LIN {X 0,Y 282.677,Z 621.959,A -85,B 0,C 180,E1 -17002.141,E2 -17002.141} C_VEL
LIN {X 0,Y 282.367,Z 625.254,A -85,B 0,C 180,E1 -17004.621,E2 -17004.621} C_VEL
LIN {X 0,Y 282.315,Z 626.398,A -85,B 0,C 180,E1 -17005.718,E2 -17005.718} C_VEL
LIN {X 0,Y 282.332,Z 627.925,A -85,B 0,C 180,E1 -17008.574,E2 -17008.574} C_VEL
LIN {X 0,Y 282.345,Z 628.204,A -85,B 0,C 180,E1 -17010,E2 -17010} C_VEL
LIN {X 0,Y 282.337,Z 627.328,A -85,B 0,C 180,E1 -17012.854,E2 -17012.854} C_VEL
LIN {X 0,Y 282.306,Z 626.397,A -85,B 0,C 180,E1 -17014.283,E2 -17014.283} C_VEL
LIN {X 0,Y 282.519,Z 623.046,A -85,B 0,C 180,E1 -17017.145,E2 -17017.145} C_VEL
LIN {X 0,Y 282.977,Z 619.419,A -85,B 0,C 180,E1 -17019.29,E2 -17019.29} C_VEL
LIN {X 0,Y 283.708,Z 614.686,A -85,B 0,C 180,E1 -17021.431,E2 -17021.431} C_VEL
LIN {X 0,Y 284.724,Z 608.712,A -85,B 0,C 180,E1 -17023.562,E2 -17023.562} C_VEL
LIN {X 0,Y 285.907,Z 602.622,A -85,B 0,C 180,E1 -17025.323,E2 -17025.323} C_VEL
LIN {X 0,Y 286.999,Z 596.881,A -85,B 0,C 180,E1 -17026.722,E2 -17026.722} C_VEL
LIN {X 0,Y 288.152,Z 590.134,A -85,B 0,C 180,E1 -17028.135,E2 -17028.135} C_VEL
LIN {X 0,Y 289.484,Z 582.394,A -85,B 0,C 180,E1 -17029.501,E2 -17029.501} C_VEL
LIN {X 0,Y 290.885,Z 574.312,A -85,B 0,C 180,E1 -17030.693,E2 -17030.693} C_VEL
LIN {X 0,Y 292.407,Z 564.552,A -85,B 0,C 180,E1 -17031.873,E2 -17031.873} C_VEL
LIN {X 0,Y 293.597,Z 556.164,A -85,B 0,C 180,E1 -17032.706,E2 -17032.706} C_VEL
LIN {X 0,Y 294.798,Z 545.658,A -85,B 0,C 180,E1 -17033.536,E2 -17033.536} C_VEL
LIN {X 0,Y 295.824,Z 535.327,A -85,B 0,C 180,E1 -17034.147,E2 -17034.147} C_VEL
LIN {X 0,Y 296.624,Z 524.607,A -85,B 0,C 180,E1 -17034.59,E2 -17034.59} C_VEL
LIN {X 0,Y 297.281,Z 501.825,A -85,B 0,C 180,E1 -17035.185,E2 -17035.185} C_VEL
LIN {X 0,Y 298.188,Z 463.102,A -85,B 0,C 180,E1 -17036.115,E2 -17036.115} C_VEL
LIN {X 0,Y 294.233,Z 440.93,A -85,B 0,C 180,E1 -17037.083,E2 -17037.083} C_VEL
LIN {X 0,Y 290.099,Z 422.604,A -85,B 0,C 180,E1 -17037.999,E2 -17037.999} C_VEL
LIN {X 0,Y 288.072,Z 417.192,A -85,B 0,C 180,E1 -17038.41,E2 -17038.41} C_VEL
LIN {X 0,Y 287.324,Z 413.003,A -85,B 0,C 180,E1 -17040.095,E2 -17040.095} C_VEL
LIN {X 0,Y 285.657,Z 404.663,A -85,B 0,C 180,E1 -17043.788,E2 -17043.788} C_VEL
LIN {X 0,Y 284.373,Z 398.634,A -85,B 0,C 180,E1 -17046.6,E2 -17046.6} C_VEL
LIN {X 0,Y 284.309,Z 398.542,A -85,B 0,C 180,E1 -17049.994,E2 -17049.994} C_VEL
LIN {X 0,Y 284.297,Z 398.571,A -85,B 0,C 180,E1 -17054.2,E2 -17054.2} C_VEL
LIN {X 0,Y 284.344,Z 398.565,A -85,B 0,C 180,E1 -17058.136,E2 -17058.136} C_VEL
LIN {X 0,Y 284.348,Z 398.566,A -85,B 0,C 180,E1 -17062.271,E2 -17062.271} C_VEL
LIN {X 0,Y 284.325,Z 398.548,A -85,B 0,C 180,E1 -17065.352,E2 -17065.352} C_VEL
LIN {X 0,Y 284.3,Z 398.57,A -85,B 0,C 180,E1 -17068.725,E2 -17068.725} C_VEL
LIN {X 0,Y 284.399,Z 398.53,A -85,B 0,C 180,E1 -17072.826,E2 -17072.826} C_VEL
LIN {X 0,Y 284.367,Z 398.56,A -85,B 0,C 180,E1 -17076.706,E2 -17076.706} C_VEL
LIN {X 0,Y 284.403,Z 398.522,A -85,B 0,C 180,E1 -17081.261,E2 -17081.261} C_VEL
LIN {X 0,Y 284.493,Z 398.54,A -85,B 0,C 180,E1 -17084.458,E2 -17084.458} C_VEL
LIN {X 0,Y 284.488,Z 398.526,A -85,B 0,C 180,E1 -17088.601,E2 -17088.601} C_VEL
LIN {X 0,Y 284.66,Z 398.486,A -85,B 0,C 180,E1 -17091.48,E2 -17091.48} C_VEL
LIN {X 0,Y 284.601,Z 398.532,A -85,B 0,C 180,E1 -17094.33,E2 -17094.33} C_VEL
LIN {X 0,Y 284.855,Z 398.478,A -85,B 0,C 180,E1 -17098.585,E2 -17098.585} C_VEL
LIN {X 0,Y 284.854,Z 398.466,A -85,B 0,C 180,E1 -17101.413,E2 -17101.413} C_VEL
LIN {X 0,Y 284.697,Z 398.513,A -85,B 0,C 180,E1 -17107.089,E2 -17107.089} C_VEL
LIN {X 0,Y 284.565,Z 398.499,A -85,B 0,C 180,E1 -17109.955,E2 -17109.955} C_VEL
LIN {X 0,Y 284.481,Z 398.548,A -85,B 0,C 180,E1 -17114.302,E2 -17114.302} C_VEL
LIN {X 0,Y 284.423,Z 398.538,A -85,B 0,C 180,E1 -17117.248,E2 -17117.248} C_VEL
LIN {X 0,Y 284.377,Z 398.533,A -85,B 0,C 180,E1 -17120.241,E2 -17120.241} C_VEL
LIN {X 0,Y 284.367,Z 398.562,A -85,B 0,C 180,E1 -17123.875,E2 -17123.875} C_VEL
LIN {X 0,Y 284.392,Z 398.532,A -85,B 0,C 180,E1 -17127.172,E2 -17127.172} C_VEL
LIN {X 0,Y 284.291,Z 398.575,A -85,B 0,C 180,E1 -17131.274,E2 -17131.274} C_VEL
LIN {X 0,Y 284.359,Z 398.544,A -85,B 0,C 180,E1 -17135.353,E2 -17135.353} C_VEL
LIN {X 0,Y 284.32,Z 398.569,A -85,B 0,C 180,E1 -17138.167,E2 -17138.167} C_VEL
LIN {X 0,Y 284.266,Z 398.568,A -85,B 0,C 180,E1 -17142.124,E2 -17142.124} C_VEL
LIN {X 0,Y 284.265,Z 398.536,A -85,B 0,C 180,E1 -17146.191,E2 -17146.191} C_VEL
LIN {X 0,Y 284.31,Z 398.537,A -85,B 0,C 180,E1 -17150.022,E2 -17150.022} C_VEL
LIN {X 0,Y 284.352,Z 398.546,A -85,B 0,C 180,E1 -17153.617,E2 -17153.617} C_VEL
LIN {X 0,Y 284.305,Z 398.553,A -85,B 0,C 180,E1 -17157.189,E2 -17157.189} C_VEL
LIN {X 0,Y 284.363,Z 398.703,A -85,B 0,C 180,E1 -17160.85,E2 -17160.85} C_VEL
LIN {X 0,Y 284.576,Z 399.615,A -85,B 0,C 180,E1 -17161.124,E2 -17161.124} C_VEL
LIN {X 0,Y 292.914,Z 415.206,A -85,B 0,C 180,E1 -17162.477,E2 -17162.477} C_VEL
LIN {X 0,Y 300.928,Z 426.438,A -85,B 0,C 180,E1 -17163.57,E2 -17163.57} C_VEL
LIN {X 0,Y 309.009,Z 435.486,A -85,B 0,C 180,E1 -17164.629,E2 -17164.629} C_VEL
LIN {X 0,Y 316.789,Z 443.826,A -85,B 0,C 180,E1 -17165.797,E2 -17165.797} C_VEL
LIN {X 0,Y 324.498,Z 451.559,A -85,B 0,C 180,E1 -17167.12,E2 -17167.12} C_VEL
LIN {X 0,Y 332.838,Z 459.453,A -85,B 0,C 180,E1 -17168.722,E2 -17168.722} C_VEL
LIN {X 0,Y 340.835,Z 466.556,A -85,B 0,C 180,E1 -17170.438,E2 -17170.438} C_VEL
LIN {X 0,Y 346.656,Z 471.215,A -85,B 0,C 180,E1 -17171.786,E2 -17171.786} C_VEL
LIN {X 0,Y 353.083,Z 476.756,A -85,B 0,C 180,E1 -17173.442,E2 -17173.442} C_VEL
LIN {X 0,Y 358.665,Z 480.934,A -85,B 0,C 180,E1 -17175.023,E2 -17175.023} C_VEL
LIN {X 0,Y 363.781,Z 485.097,A -85,B 0,C 180,E1 -17176.663,E2 -17176.663} C_VEL
LIN {X 0,Y 368.607,Z 488.107,A -85,B 0,C 180,E1 -17178.392,E2 -17178.392} C_VEL
LIN {X 0,Y 370.69,Z 489.608,A -85,B 0,C 180,E1 -17179.248,E2 -17179.248} C_VEL
LIN {X 0,Y 374.454,Z 492.817,A -85,B 0,C 180,E1 -17181.024,E2 -17181.024} C_VEL
LIN {X 0,Y 377.635,Z 494.931,A -85,B 0,C 180,E1 -17182.837,E2 -17182.837} C_VEL
LIN {X 0,Y 380.182,Z 496.242,A -85,B 0,C 180,E1 -17184.696,E2 -17184.696} C_VEL
LIN {X 0,Y 381.691,Z 496.803,A -85,B 0,C 180,E1 -17186.149,E2 -17186.149} C_VEL
LIN {X 0,Y 382.967,Z 497.365,A -85,B 0,C 180,E1 -17188.159,E2 -17188.159} C_VEL
LIN {X 0,Y 383.351,Z 497.509,A -85,B 0,C 180,E1 -17190,E2 -17190} C_VEL
LIN {X 0,Y 383.049,Z 497.433,A -85,B 0,C 180,E1 -17191.577,E2 -17191.577} C_VEL
LIN {X 0,Y 382.23,Z 496.941,A -85,B 0,C 180,E1 -17193.162,E2 -17193.162} C_VEL
LIN {X 0,Y 380.5,Z 496.432,A -85,B 0,C 180,E1 -17195.024,E2 -17195.024} C_VEL
LIN {X 0,Y 377.946,Z 495.11,A -85,B 0,C 180,E1 -17196.961,E2 -17196.961} C_VEL
LIN {X 0,Y 374.623,Z 492.956,A -85,B 0,C 180,E1 -17198.885,E2 -17198.885} C_VEL
LIN {X 0,Y 371.032,Z 489.898,A -85,B 0,C 180,E1 -17200.604,E2 -17200.604} C_VEL
LIN {X 0,Y 368.789,Z 488.206,A -85,B 0,C 180,E1 -17201.535,E2 -17201.535} C_VEL
LIN {X 0,Y 364.031,Z 485.266,A -85,B 0,C 180,E1 -17203.256,E2 -17203.256} C_VEL
LIN {X 0,Y 358.883,Z 481.111,A -85,B 0,C 180,E1 -17204.909,E2 -17204.909} C_VEL
LIN {X 0,Y 352.314,Z 476.156,A -85,B 0,C 180,E1 -17206.765,E2 -17206.765} C_VEL
LIN {X 0,Y 345.31,Z 470.262,A -85,B 0,C 180,E1 -17208.53,E2 -17208.53} C_VEL
LIN {X 0,Y 338.898,Z 464.788,A -85,B 0,C 180,E1 -17210.001,E2 -17210.001} C_VEL
LIN {X 0,Y 331.392,Z 458.055,A -85,B 0,C 180,E1 -17211.572,E2 -17211.572} C_VEL
LIN {X 0,Y 323.341,Z 450.352,A -85,B 0,C 180,E1 -17213.096,E2 -17213.096} C_VEL
LIN {X 0,Y 316.278,Z 443.247,A -85,B 0,C 180,E1 -17214.282,E2 -17214.282} C_VEL
LIN {X 0,Y 308.675,Z 435.183,A -85,B 0,C 180,E1 -17215.413,E2 -17215.413} C_VEL
LIN {X 0,Y 300.726,Z 426.19,A -85,B 0,C 180,E1 -17216.456,E2 -17216.456} C_VEL
LIN {X 0,Y 292.805,Z 415.042,A -85,B 0,C 180,E1 -17217.539,E2 -17217.539} C_VEL
LIN {X 0,Y 284.576,Z 399.626,A -85,B 0,C 180,E1 -17218.876,E2 -17218.876} C_VEL
LIN {X 0,Y 284.351,Z 398.628,A -85,B 0,C 180,E1 -17219.189,E2 -17219.189} C_VEL
LIN {X 0,Y 284.3,Z 398.551,A -85,B 0,C 180,E1 -17222.945,E2 -17222.945} C_VEL
LIN {X 0,Y 284.35,Z 398.546,A -85,B 0,C 180,E1 -17226.382,E2 -17226.382} C_VEL
LIN {X 0,Y 284.306,Z 398.537,A -85,B 0,C 180,E1 -17229.993,E2 -17229.993} C_VEL
LIN {X 0,Y 284.259,Z 398.545,A -85,B 0,C 180,E1 -17234.195,E2 -17234.195} C_VEL
LIN {X 0,Y 284.296,Z 398.561,A -85,B 0,C 180,E1 -17238.13,E2 -17238.13} C_VEL
LIN {X 0,Y 284.328,Z 398.568,A -85,B 0,C 180,E1 -17241.835,E2 -17241.835} C_VEL
LIN {X 0,Y 284.317,Z 398.546,A -85,B 0,C 180,E1 -17245.353,E2 -17245.353} C_VEL
LIN {X 0,Y 284.29,Z 398.575,A -85,B 0,C 180,E1 -17248.726,E2 -17248.726} C_VEL
LIN {X 0,Y 284.391,Z 398.533,A -85,B 0,C 180,E1 -17252.827,E2 -17252.827} C_VEL
LIN {X 0,Y 284.36,Z 398.564,A -85,B 0,C 180,E1 -17256.707,E2 -17256.707} C_VEL
LIN {X 0,Y 284.397,Z 398.526,A -85,B 0,C 180,E1 -17261.262,E2 -17261.262} C_VEL
LIN {X 0,Y 284.486,Z 398.547,A -85,B 0,C 180,E1 -17264.46,E2 -17264.46} C_VEL
LIN {X 0,Y 284.484,Z 398.519,A -85,B 0,C 180,E1 -17268.602,E2 -17268.602} C_VEL
LIN {X 0,Y 284.654,Z 398.501,A -85,B 0,C 180,E1 -17271.482,E2 -17271.482} C_VEL
LIN {X 0,Y 284.597,Z 398.534,A -85,B 0,C 180,E1 -17274.332,E2 -17274.332} C_VEL
LIN {X 0,Y 284.851,Z 398.466,A -85,B 0,C 180,E1 -17278.587,E2 -17278.587} C_VEL
LIN {X 0,Y 284.851,Z 398.478,A -85,B 0,C 180,E1 -17281.415,E2 -17281.415} C_VEL
LIN {X 0,Y 284.694,Z 398.507,A -85,B 0,C 180,E1 -17287.091,E2 -17287.091} C_VEL
LIN {X 0,Y 284.562,Z 398.498,A -85,B 0,C 180,E1 -17289.956,E2 -17289.956} C_VEL
LIN {X 0,Y 284.478,Z 398.547,A -85,B 0,C 180,E1 -17294.304,E2 -17294.304} C_VEL
LIN {X 0,Y 284.422,Z 398.527,A -85,B 0,C 180,E1 -17297.249,E2 -17297.249} C_VEL
LIN {X 0,Y 284.38,Z 398.535,A -85,B 0,C 180,E1 -17300.007,E2 -17300.007} C_VEL
LIN {X 0,Y 283.742,Z 398.633,A -85,B 0,C 180,E1 -17301.19,E2 -17301.19} C_VEL
LIN {X 0,Y 280.865,Z 398.996,A -85,B 0,C 180,E1 -17303.115,E2 -17303.115} C_VEL
LIN {X 0,Y 278.413,Z 399.292,A -85,B 0,C 180,E1 -17304.68,E2 -17304.68} C_VEL
LIN {X 0,Y 277.379,Z 399.406,A -85,B 0,C 180,E1 -17305.893,E2 -17305.893} C_VEL
LIN {X 0,Y 277.306,Z 399.412,A -85,B 0,C 180,E1 -17306.304,E2 -17306.304} C_VEL
LIN {X 0,Y 277.27,Z 399.448,A -85,B 0,C 180,E1 -17310.483,E2 -17310.483} C_VEL
LIN {X 0,Y 277.253,Z 399.426,A -85,B 0,C 180,E1 -17313.896,E2 -17313.896} C_VEL
LIN {X 0,Y 277.29,Z 399.445,A -85,B 0,C 180,E1 -17317.467,E2 -17317.467} C_VEL
LIN {X 0,Y 277.293,Z 399.44,A -85,B 0,C 180,E1 -17321.222,E2 -17321.222} C_VEL
LIN {X 0,Y 277.242,Z 399.446,A -85,B 0,C 180,E1 -17325.219,E2 -17325.219} C_VEL
LIN {X 0,Y 277.225,Z 399.422,A -85,B 0,C 180,E1 -17329.513,E2 -17329.513} C_VEL
LIN {X 0,Y 277.332,Z 399.542,A -85,B 0,C 180,E1 -17332.853,E2 -17332.853} C_VEL
LIN {X 0,Y 278.869,Z 406.848,A -85,B 0,C 180,E1 -17336.329,E2 -17336.329} C_VEL
LIN {X 0,Y 280.483,Z 414.722,A -85,B 0,C 180,E1 -17339.926,E2 -17339.926} C_VEL
LIN {X 0,Y 280.854,Z 417.027,A -85,B 0,C 180,E1 -17340.797,E2 -17340.797} C_VEL
LIN {X 0,Y 284.61,Z 426.762,A -85,B 0,C 180,E1 -17341.534,E2 -17341.534} C_VEL
LIN {X 0,Y 289.763,Z 451.78,A -85,B 0,C 180,E1 -17342.764,E2 -17342.764} C_VEL
LIN {X 0,Y 291.922,Z 464.944,A -85,B 0,C 180,E1 -17343.335,E2 -17343.335} C_VEL
LIN {X 0,Y 290.246,Z 521.874,A -85,B 0,C 180,E1 -17344.738,E2 -17344.738} C_VEL
LIN {X 0,Y 289.59,Z 532.566,A -85,B 0,C 180,E1 -17345.157,E2 -17345.157} C_VEL
LIN {X 0,Y 288.57,Z 542.95,A -85,B 0,C 180,E1 -17345.734,E2 -17345.734} C_VEL
LIN {X 0,Y 287.511,Z 552.041,A -85,B 0,C 180,E1 -17346.405,E2 -17346.405} C_VEL
LIN {X 0,Y 286.343,Z 561.187,A -85,B 0,C 180,E1 -17347.26,E2 -17347.26} C_VEL
LIN {X 0,Y 284.896,Z 570.185,A -85,B 0,C 180,E1 -17348.283,E2 -17348.283} C_VEL
LIN {X 0,Y 283.35,Z 578.908,A -85,B 0,C 180,E1 -17349.492,E2 -17349.492} C_VEL
LIN {X 0,Y 281.997,Z 586.328,A -85,B 0,C 180,E1 -17350.719,E2 -17350.719} C_VEL
LIN {X 0,Y 280.585,Z 594.399,A -85,B 0,C 180,E1 -17352.333,E2 -17352.333} C_VEL
LIN {X 0,Y 279.266,Z 601.116,A -85,B 0,C 180,E1 -17353.93,E2 -17353.93} C_VEL
LIN {X 0,Y 278.03,Z 607.427,A -85,B 0,C 180,E1 -17355.733,E2 -17355.733} C_VEL
LIN {X 0,Y 276.988,Z 612.7,A -85,B 0,C 180,E1 -17357.546,E2 -17357.546} C_VEL
LIN {X 0,Y 276.17,Z 617.796,A -85,B 0,C 180,E1 -17359.739,E2 -17359.739} C_VEL
LIN {X 0,Y 275.606,Z 621.763,A -85,B 0,C 180,E1 -17361.938,E2 -17361.938} C_VEL
LIN {X 0,Y 275.257,Z 625.322,A -85,B 0,C 180,E1 -17364.734,E2 -17364.734} C_VEL
LIN {X 0,Y 275.229,Z 626.202,A -85,B 0,C 180,E1 -17365.607,E2 -17365.607} C_VEL
LIN {X 0,Y 275.256,Z 627.73,A -85,B 0,C 180,E1 -17368.537,E2 -17368.537} C_VEL
LIN {X 0,Y 275.267,Z 628.01,A -85,B 0,C 180,E1 -17370,E2 -17370} C_VEL
LIN {X 0,Y 275.246,Z 627.133,A -85,B 0,C 180,E1 -17372.928,E2 -17372.928} C_VEL
LIN {X 0,Y 275.241,Z 625.361,A -85,B 0,C 180,E1 -17375.229,E2 -17375.229} C_VEL
LIN {X 0,Y 275.607,Z 621.762,A -85,B 0,C 180,E1 -17378.063,E2 -17378.063} C_VEL
LIN {X 0,Y 276.171,Z 617.795,A -85,B 0,C 180,E1 -17380.262,E2 -17380.262} C_VEL
LIN {X 0,Y 276.986,Z 612.697,A -85,B 0,C 180,E1 -17382.455,E2 -17382.455} C_VEL
LIN {X 0,Y 278.537,Z 605.049,A -85,B 0,C 180,E1 -17384.989,E2 -17384.989} C_VEL
LIN {X 0,Y 279.872,Z 598.245,A -85,B 0,C 180,E1 -17386.785,E2 -17386.785} C_VEL
LIN {X 0,Y 281.304,Z 590.341,A -85,B 0,C 180,E1 -17388.511,E2 -17388.511} C_VEL
LIN {X 0,Y 282.788,Z 582.198,A -85,B 0,C 180,E1 -17389.982,E2 -17389.982} C_VEL
LIN {X 0,Y 284.237,Z 574.116,A -85,B 0,C 180,E1 -17391.2,E2 -17391.2} C_VEL
LIN {X 0,Y 285.827,Z 564.357,A -85,B 0,C 180,E1 -17392.403,E2 -17392.403} C_VEL
LIN {X 0,Y 287.038,Z 555.968,A -85,B 0,C 180,E1 -17393.254,E2 -17393.254} C_VEL
LIN {X 0,Y 288.296,Z 545.462,A -85,B 0,C 180,E1 -17394.1,E2 -17394.1} C_VEL
LIN {X 0,Y 289.357,Z 535.132,A -85,B 0,C 180,E1 -17394.722,E2 -17394.722} C_VEL
LIN {X 0,Y 290.172,Z 524.412,A -85,B 0,C 180,E1 -17395.174,E2 -17395.174} C_VEL
LIN {X 0,Y 290.884,Z 500.338,A -85,B 0,C 180,E1 -17395.813,E2 -17395.813} C_VEL
LIN {X 0,Y 291.82,Z 464.357,A -85,B 0,C 180,E1 -17396.691,E2 -17396.691} C_VEL
LIN {X 0,Y 288.064,Z 442.873,A -85,B 0,C 180,E1 -17397.653,E2 -17397.653} C_VEL
LIN {X 0,Y 284.148,Z 425.282,A -85,B 0,C 180,E1 -17398.558,E2 -17398.558} C_VEL
LIN {X 0,Y 280.871,Z 416.937,A -85,B 0,C 180,E1 -17399.213,E2 -17399.213} C_VEL
LIN {X 0,Y 279.698,Z 410.828,A -85,B 0,C 180,E1 -17401.848,E2 -17401.848} C_VEL
LIN {X 0,Y 277.859,Z 401.977,A -85,B 0,C 180,E1 -17405.962,E2 -17405.962} C_VEL
LIN {X 0,Y 277.324,Z 399.495,A -85,B 0,C 180,E1 -17407.253,E2 -17407.253} C_VEL
LIN {X 0,Y 277.218,Z 399.423,A -85,B 0,C 180,E1 -17411.235,E2 -17411.235} C_VEL
LIN {X 0,Y 277.249,Z 399.441,A -85,B 0,C 180,E1 -17415.216,E2 -17415.216} C_VEL
LIN {X 0,Y 277.298,Z 399.431,A -85,B 0,C 180,E1 -17419.494,E2 -17419.494} C_VEL
LIN {X 0,Y 277.293,Z 399.445,A -85,B 0,C 180,E1 -17422.534,E2 -17422.534} C_VEL
LIN {X 0,Y 277.256,Z 399.425,A -85,B 0,C 180,E1 -17426.105,E2 -17426.105} C_VEL
LIN {X 0,Y 277.263,Z 399.449,A -85,B 0,C 180,E1 -17429.538,E2 -17429.538} C_VEL
LIN {X 0,Y 277.36,Z 399.406,A -85,B 0,C 180,E1 -17432.863,E2 -17432.863} C_VEL
LIN {X 0,Y 277.33,Z 399.434,A -85,B 0,C 180,E1 -17436.079,E2 -17436.079} C_VEL
LIN {X 0,Y 277.345,Z 399.403,A -85,B 0,C 180,E1 -17440.765,E2 -17440.765} C_VEL
LIN {X 0,Y 277.435,Z 399.422,A -85,B 0,C 180,E1 -17445.325,E2 -17445.325} C_VEL
LIN {X 0,Y 277.507,Z 399.376,A -85,B 0,C 180,E1 -17449.788,E2 -17449.788} C_VEL
LIN {X 0,Y 277.653,Z 399.378,A -85,B 0,C 180,E1 -17452.728,E2 -17452.728} C_VEL
LIN {X 0,Y 277.821,Z 399.353,A -85,B 0,C 180,E1 -17458.55,E2 -17458.55} C_VEL
LIN {X 0,Y 277.82,Z 399.342,A -85,B 0,C 180,E1 -17461.449,E2 -17461.449} C_VEL
LIN {X 0,Y 277.652,Z 399.387,A -85,B 0,C 180,E1 -17467.27,E2 -17467.27} C_VEL
LIN {X 0,Y 277.506,Z 399.378,A -85,B 0,C 180,E1 -17470.21,E2 -17470.21} C_VEL
LIN {X 0,Y 277.433,Z 399.426,A -85,B 0,C 180,E1 -17474.673,E2 -17474.673} C_VEL
LIN {X 0,Y 277.343,Z 399.403,A -85,B 0,C 180,E1 -17479.233,E2 -17479.233} C_VEL
LIN {X 0,Y 277.317,Z 399.439,A -85,B 0,C 180,E1 -17484.169,E2 -17484.169} C_VEL
LIN {X 0,Y 277.321,Z 399.412,A -85,B 0,C 180,E1 -17487.503,E2 -17487.503} C_VEL
LIN {X 0,Y 277.269,Z 399.446,A -85,B 0,C 180,E1 -17490.481,E2 -17490.481} C_VEL
LIN {X 0,Y 277.251,Z 399.428,A -85,B 0,C 180,E1 -17493.894,E2 -17493.894} C_VEL
LIN {X 0,Y 277.279,Z 399.448,A -85,B 0,C 180,E1 -17497.466,E2 -17497.466} C_VEL
LIN {X 0,Y 277.207,Z 399.438,A -85,B 0,C 180,E1 -17501.236,E2 -17501.236} C_VEL
LIN {X 0,Y 277.213,Z 399.436,A -85,B 0,C 180,E1 -17505.223,E2 -17505.223} C_VEL
LIN {X 0,Y 277.224,Z 399.408,A -85,B 0,C 180,E1 -17509.51,E2 -17509.51} C_VEL
LIN {X 0,Y 277.287,Z 399.445,A -85,B 0,C 180,E1 -17512.534,E2 -17512.534} C_VEL
LIN {X 0,Y 277.251,Z 399.416,A -85,B 0,C 180,E1 -17516.105,E2 -17516.105} C_VEL
LIN {X 0,Y 277.31,Z 399.572,A -85,B 0,C 180,E1 -17520.071,E2 -17520.071} C_VEL
LIN {X 0,Y 277.562,Z 400.54,A -85,B 0,C 180,E1 -17520.346,E2 -17520.346} C_VEL
LIN {X 0,Y 287.682,Z 419.481,A -85,B 0,C 180,E1 -17522.047,E2 -17522.047} C_VEL
LIN {X 0,Y 295.526,Z 430.618,A -85,B 0,C 180,E1 -17523.156,E2 -17523.156} C_VEL
LIN {X 0,Y 304.61,Z 440.791,A -85,B 0,C 180,E1 -17524.305,E2 -17524.305} C_VEL
LIN {X 0,Y 311.067,Z 447.49,A -85,B 0,C 180,E1 -17525.192,E2 -17525.192} C_VEL
LIN {X 0,Y 317.093,Z 453.543,A -85,B 0,C 180,E1 -17526.104,E2 -17526.104} C_VEL
LIN {X 0,Y 324.326,Z 460.47,A -85,B 0,C 180,E1 -17527.35,E2 -17527.35} C_VEL
LIN {X 0,Y 332.422,Z 467.895,A -85,B 0,C 180,E1 -17528.905,E2 -17528.905} C_VEL
LIN {X 0,Y 340.798,Z 475.078,A -85,B 0,C 180,E1 -17530.702,E2 -17530.702} C_VEL
LIN {X 0,Y 346.857,Z 479.951,A -85,B 0,C 180,E1 -17532.123,E2 -17532.123} C_VEL
LIN {X 0,Y 352.732,Z 484.601,A -85,B 0,C 180,E1 -17533.635,E2 -17533.635} C_VEL
LIN {X 0,Y 356.978,Z 487.769,A -85,B 0,C 180,E1 -17534.83,E2 -17534.83} C_VEL
LIN {X 0,Y 362.245,Z 491.918,A -85,B 0,C 180,E1 -17536.484,E2 -17536.484} C_VEL
LIN {X 0,Y 366.997,Z 494.884,A -85,B 0,C 180,E1 -17538.151,E2 -17538.151} C_VEL
LIN {X 0,Y 369.342,Z 496.523,A -85,B 0,C 180,E1 -17539.083,E2 -17539.083} C_VEL
LIN {X 0,Y 373.181,Z 499.677,A -85,B 0,C 180,E1 -17540.846,E2 -17540.846} C_VEL
LIN {X 0,Y 376.178,Z 501.679,A -85,B 0,C 180,E1 -17542.485,E2 -17542.485} C_VEL
LIN {X 0,Y 378.846,Z 503.096,A -85,B 0,C 180,E1 -17544.299,E2 -17544.299} C_VEL
LIN {X 0,Y 380.516,Z 503.759,A -85,B 0,C 180,E1 -17545.826,E2 -17545.826} C_VEL
LIN {X 0,Y 381.686,Z 504.194,A -85,B 0,C 180,E1 -17547.349,E2 -17547.349} C_VEL
LIN {X 0,Y 382.346,Z 504.597,A -85,B 0,C 180,E1 -17548.946,E2 -17548.946} C_VEL
LIN {X 0,Y 382.487,Z 504.54,A -85,B 0,C 180,E1 -17550,E2 -17550} C_VEL
LIN {X 0,Y 382.181,Z 504.482,A -85,B 0,C 180,E1 -17551.58,E2 -17551.58} C_VEL
LIN {X 0,Y 381.353,Z 503.983,A -85,B 0,C 180,E1 -17553.169,E2 -17553.169} C_VEL
LIN {X 0,Y 379.487,Z 503.421,A -85,B 0,C 180,E1 -17555.14,E2 -17555.14} C_VEL
LIN {X 0,Y 376.716,Z 501.958,A -85,B 0,C 180,E1 -17557.182,E2 -17557.182} C_VEL
LIN {X 0,Y 373.349,Z 499.834,A -85,B 0,C 180,E1 -17559.071,E2 -17559.071} C_VEL
LIN {X 0,Y 369.653,Z 496.798,A -85,B 0,C 180,E1 -17560.785,E2 -17560.785} C_VEL
LIN {X 0,Y 367.139,Z 494.937,A -85,B 0,C 180,E1 -17561.798,E2 -17561.798} C_VEL
LIN {X 0,Y 362.574,Z 492.144,A -85,B 0,C 180,E1 -17563.407,E2 -17563.407} C_VEL
LIN {X 0,Y 356.978,Z 487.768,A -85,B 0,C 180,E1 -17565.17,E2 -17565.17} C_VEL
LIN {X 0,Y 350.018,Z 482.598,A -85,B 0,C 180,E1 -17567.073,E2 -17567.073} C_VEL
LIN {X 0,Y 342.612,Z 476.491,A -85,B 0,C 180,E1 -17568.893,E2 -17568.893} C_VEL
LIN {X 0,Y 335.883,Z 470.825,A -85,B 0,C 180,E1 -17570.376,E2 -17570.376} C_VEL
LIN {X 0,Y 328.346,Z 464.224,A -85,B 0,C 180,E1 -17571.902,E2 -17571.902} C_VEL
LIN {X 0,Y 319.943,Z 456.342,A -85,B 0,C 180,E1 -17573.421,E2 -17573.421} C_VEL
LIN {X 0,Y 312.094,Z 448.619,A -85,B 0,C 180,E1 -17574.656,E2 -17574.656} C_VEL
LIN {X 0,Y 304.274,Z 440.475,A -85,B 0,C 180,E1 -17575.738,E2 -17575.738} C_VEL
LIN {X 0,Y 294.922,Z 429.801,A -85,B 0,C 180,E1 -17576.926,E2 -17576.926} C_VEL
LIN {X 0,Y 287.345,Z 418.928,A -85,B 0,C 180,E1 -17578.004,E2 -17578.004} C_VEL
LIN {X 0,Y 277.552,Z 400.569,A -85,B 0,C 180,E1 -17579.65,E2 -17579.65} C_VEL
LIN {X 0,Y 277.303,Z 399.52,A -85,B 0,C 180,E1 -17579.965,E2 -17579.965} C_VEL
LIN {X 0,Y 277.249,Z 399.416,A -85,B 0,C 180,E1 -17583.894,E2 -17583.894} C_VEL
LIN {X 0,Y 277.285,Z 399.445,A -85,B 0,C 180,E1 -17587.465,E2 -17587.465} C_VEL
LIN {X 0,Y 277.206,Z 399.401,A -85,B 0,C 180,E1 -17591.236,E2 -17591.236} C_VEL
LIN {X 0,Y 277.218,Z 399.442,A -85,B 0,C 180,E1 -17595.222,E2 -17595.222} C_VEL
LIN {X 0,Y 277.256,Z 399.431,A -85,B 0,C 180,E1 -17599.503,E2 -17599.503} C_VEL
LIN {X 0,Y 277.284,Z 399.448,A -85,B 0,C 180,E1 -17602.534,E2 -17602.534} C_VEL
LIN {X 0,Y 277.248,Z 399.428,A -85,B 0,C 180,E1 -17606.106,E2 -17606.106} C_VEL
LIN {X 0,Y 277.255,Z 399.448,A -85,B 0,C 180,E1 -17609.539,E2 -17609.539} C_VEL
LIN {X 0,Y 277.353,Z 399.409,A -85,B 0,C 180,E1 -17612.864,E2 -17612.864} C_VEL
LIN {X 0,Y 277.323,Z 399.439,A -85,B 0,C 180,E1 -17616.08,E2 -17616.08} C_VEL
LIN {X 0,Y 277.339,Z 399.403,A -85,B 0,C 180,E1 -17620.767,E2 -17620.767} C_VEL
LIN {X 0,Y 277.429,Z 399.426,A -85,B 0,C 180,E1 -17625.326,E2 -17625.326} C_VEL
LIN {X 0,Y 277.502,Z 399.378,A -85,B 0,C 180,E1 -17629.789,E2 -17629.789} C_VEL
LIN {X 0,Y 277.648,Z 399.388,A -85,B 0,C 180,E1 -17632.73,E2 -17632.73} C_VEL
LIN {X 0,Y 277.817,Z 399.342,A -85,B 0,C 180,E1 -17638.551,E2 -17638.551} C_VEL
LIN {X 0,Y 277.817,Z 399.354,A -85,B 0,C 180,E1 -17641.45,E2 -17641.45} C_VEL
LIN {X 0,Y 277.649,Z 399.379,A -85,B 0,C 180,E1 -17647.272,E2 -17647.272} C_VEL
LIN {X 0,Y 277.503,Z 399.378,A -85,B 0,C 180,E1 -17650.212,E2 -17650.212} C_VEL
LIN {X 0,Y 277.431,Z 399.422,A -85,B 0,C 180,E1 -17654.675,E2 -17654.675} C_VEL
LIN {X 0,Y 277.341,Z 399.403,A -85,B 0,C 180,E1 -17659.235,E2 -17659.235} C_VEL
LIN {X 0,Y 277.316,Z 399.432,A -85,B 0,C 180,E1 -17664.171,E2 -17664.171} C_VEL
LIN {X 0,Y 277.306,Z 399.412,A -85,B 0,C 180,E1 -17666.304,E2 -17666.304} C_VEL
LIN {X 0,Y 276.646,Z 399.499,A -85,B 0,C 180,E1 -17667.516,E2 -17667.516} C_VEL
LIN {X 0,Y 273.729,Z 399.884,A -85,B 0,C 180,E1 -17669.488,E2 -17669.488} C_VEL
LIN {X 0,Y 271.263,Z 400.194,A -85,B 0,C 180,E1 -17671.091,E2 -17671.091} C_VEL
LIN {X 0,Y 270.242,Z 400.31,A -85,B 0,C 180,E1 -17672.336,E2 -17672.336} C_VEL
LIN {X 0,Y 270.179,Z 400.311,A -85,B 0,C 180,E1 -17672.758,E2 -17672.758} C_VEL
LIN {X 0,Y 270.242,Z 400.323,A -85,B 0,C 180,E1 -17676.738,E2 -17676.738} C_VEL
LIN {X 0,Y 270.267,Z 400.312,A -85,B 0,C 180,E1 -17681.054,E2 -17681.054} C_VEL
LIN {X 0,Y 270.189,Z 400.326,A -85,B 0,C 180,E1 -17685.389,E2 -17685.389} C_VEL
LIN {X 0,Y 270.177,Z 400.299,A -85,B 0,C 180,E1 -17689.436,E2 -17689.436} C_VEL
LIN {X 0,Y 270.276,Z 400.487,A -85,B 0,C 180,E1 -17692.275,E2 -17692.275} C_VEL
LIN {X 0,Y 271.822,Z 407.725,A -85,B 0,C 180,E1 -17695.83,E2 -17695.83} C_VEL
LIN {X 0,Y 273.594,Z 416.41,A -85,B 0,C 180,E1 -17699.859,E2 -17699.859} C_VEL
LIN {X 0,Y 274.024,Z 417.952,A -85,B 0,C 180,E1 -17700.066,E2 -17700.066} C_VEL
LIN {X 0,Y 278.637,Z 429.273,A -85,B 0,C 180,E1 -17700.943,E2 -17700.943} C_VEL
LIN {X 0,Y 283.558,Z 453.545,A -85,B 0,C 180,E1 -17702.172,E2 -17702.172} C_VEL
LIN {X 0,Y 285.556,Z 465.963,A -85,B 0,C 180,E1 -17702.726,E2 -17702.726} C_VEL
LIN {X 0,Y 283.856,Z 521.686,A -85,B 0,C 180,E1 -17704.128,E2 -17704.128} C_VEL
LIN {X 0,Y 283.174,Z 532.372,A -85,B 0,C 180,E1 -17704.554,E2 -17704.554} C_VEL
LIN {X 0,Y 282.103,Z 542.755,A -85,B 0,C 180,E1 -17705.141,E2 -17705.141} C_VEL
LIN {X 0,Y 281.015,Z 551.846,A -85,B 0,C 180,E1 -17705.826,E2 -17705.826} C_VEL
LIN {X 0,Y 279.803,Z 560.991,A -85,B 0,C 180,E1 -17706.697,E2 -17706.697} C_VEL
LIN {X 0,Y 278.289,Z 569.989,A -85,B 0,C 180,E1 -17707.741,E2 -17707.741} C_VEL
LIN {X 0,Y 276.699,Z 578.713,A -85,B 0,C 180,E1 -17708.976,E2 -17708.976} C_VEL
LIN {X 0,Y 275.296,Z 586.132,A -85,B 0,C 180,E1 -17710.23,E2 -17710.23} C_VEL
LIN {X 0,Y 273.893,Z 593.442,A -85,B 0,C 180,E1 -17711.699,E2 -17711.699} C_VEL
LIN {X 0,Y 272.416,Z 600.92,A -85,B 0,C 180,E1 -17713.514,E2 -17713.514} C_VEL
LIN {X 0,Y 271.125,Z 607.231,A -85,B 0,C 180,E1 -17715.361,E2 -17715.361} C_VEL
LIN {X 0,Y 270.028,Z 612.504,A -85,B 0,C 180,E1 -17717.219,E2 -17717.219} C_VEL
LIN {X 0,Y 269.158,Z 617.601,A -85,B 0,C 180,E1 -17719.469,E2 -17719.469} C_VEL
LIN {X 0,Y 268.553,Z 621.567,A -85,B 0,C 180,E1 -17721.725,E2 -17721.725} C_VEL
LIN {X 0,Y 268.169,Z 625.341,A -85,B 0,C 180,E1 -17724.804,E2 -17724.804} C_VEL
LIN {X 0,Y 268.16,Z 626.939,A -85,B 0,C 180,E1 -17726.996,E2 -17726.996} C_VEL
LIN {X 0,Y 268.192,Z 627.816,A -85,B 0,C 180,E1 -17730,E2 -17730} C_VEL
LIN {X 0,Y 268.157,Z 626.938,A -85,B 0,C 180,E1 -17733.005,E2 -17733.005} C_VEL
LIN {X 0,Y 268.166,Z 625.348,A -85,B 0,C 180,E1 -17735.188,E2 -17735.188} C_VEL
LIN {X 0,Y 268.553,Z 621.566,A -85,B 0,C 180,E1 -17738.276,E2 -17738.276} C_VEL
LIN {X 0,Y 269.159,Z 617.599,A -85,B 0,C 180,E1 -17740.532,E2 -17740.532} C_VEL
LIN {X 0,Y 270.026,Z 612.502,A -85,B 0,C 180,E1 -17742.782,E2 -17742.782} C_VEL
LIN {X 0,Y 271.67,Z 604.854,A -85,B 0,C 180,E1 -17745.377,E2 -17745.377} C_VEL
LIN {X 0,Y 273.074,Z 598.05,A -85,B 0,C 180,E1 -17747.216,E2 -17747.216} C_VEL
LIN {X 0,Y 274.63,Z 589.835,A -85,B 0,C 180,E1 -17749.042,E2 -17749.042} C_VEL
LIN {X 0,Y 276.09,Z 582.002,A -85,B 0,C 180,E1 -17750.488,E2 -17750.488} C_VEL
LIN {X 0,Y 277.609,Z 573.921,A -85,B 0,C 180,E1 -17751.731,E2 -17751.731} C_VEL
LIN {X 0,Y 279.262,Z 564.162,A -85,B 0,C 180,E1 -17752.959,E2 -17752.959} C_VEL
LIN {X 0,Y 280.519,Z 555.773,A -85,B 0,C 180,E1 -17753.828,E2 -17753.828} C_VEL
LIN {X 0,Y 281.821,Z 545.267,A -85,B 0,C 180,E1 -17754.69,E2 -17754.69} C_VEL
LIN {X 0,Y 282.924,Z 534.936,A -85,B 0,C 180,E1 -17755.323,E2 -17755.323} C_VEL
LIN {X 0,Y 283.768,Z 524.217,A -85,B 0,C 180,E1 -17755.783,E2 -17755.783} C_VEL
LIN {X 0,Y 284.503,Z 500.303,A -85,B 0,C 180,E1 -17756.432,E2 -17756.432} C_VEL
LIN {X 0,Y 285.403,Z 464.794,A -85,B 0,C 180,E1 -17757.322,E2 -17757.322} C_VEL
LIN {X 0,Y 281.736,Z 444.013,A -85,B 0,C 180,E1 -17758.292,E2 -17758.292} C_VEL
LIN {X 0,Y 278.315,Z 428.226,A -85,B 0,C 180,E1 -17759.123,E2 -17759.123} C_VEL
LIN {X 0,Y 273.692,Z 416.944,A -85,B 0,C 180,E1 -17760.027,E2 -17760.027} C_VEL
LIN {X 0,Y 273.514,Z 416.127,A -85,B 0,C 180,E1 -17760.241,E2 -17760.241} C_VEL
LIN {X 0,Y 271.837,Z 407.711,A -85,B 0,C 180,E1 -17764.174,E2 -17764.174} C_VEL
LIN {X 0,Y 270.27,Z 400.408,A -85,B 0,C 180,E1 -17767.786,E2 -17767.786} C_VEL
LIN {X 0,Y 270.19,Z 400.314,A -85,B 0,C 180,E1 -17772.555,E2 -17772.555} C_VEL
LIN {X 0,Y 270.216,Z 400.321,A -85,B 0,C 180,E1 -17776.74,E2 -17776.74} C_VEL
LIN {X 0,Y 270.251,Z 400.309,A -85,B 0,C 180,E1 -17779.447,E2 -17779.447} C_VEL
LIN {X 0,Y 270.26,Z 400.316,A -85,B 0,C 180,E1 -17783.72,E2 -17783.72} C_VEL
LIN {X 0,Y 270.207,Z 400.306,A -85,B 0,C 180,E1 -17786.892,E2 -17786.892} C_VEL
LIN {X 0,Y 270.231,Z 400.32,A -85,B 0,C 180,E1 -17790.386,E2 -17790.386} C_VEL
LIN {X 0,Y 270.265,Z 400.289,A -85,B 0,C 180,E1 -17793.763,E2 -17793.763} C_VEL
LIN {X 0,Y 270.234,Z 400.32,A -85,B 0,C 180,E1 -17797.038,E2 -17797.038} C_VEL
LIN {X 0,Y 270.302,Z 400.285,A -85,B 0,C 180,E1 -17800.244,E2 -17800.244} C_VEL
LIN {X 0,Y 270.403,Z 400.296,A -85,B 0,C 180,E1 -17804.935,E2 -17804.935} C_VEL
LIN {X 0,Y 270.442,Z 400.258,A -85,B 0,C 180,E1 -17809.518,E2 -17809.518} C_VEL
LIN {X 0,Y 270.611,Z 400.25,A -85,B 0,C 180,E1 -17812.538,E2 -17812.538} C_VEL
LIN {X 0,Y 270.787,Z 400.229,A -85,B 0,C 180,E1 -17818.512,E2 -17818.512} C_VEL
LIN {X 0,Y 270.786,Z 400.217,A -85,B 0,C 180,E1 -17821.486,E2 -17821.486} C_VEL
LIN {X 0,Y 270.61,Z 400.262,A -85,B 0,C 180,E1 -17827.46,E2 -17827.46} C_VEL
LIN {X 0,Y 270.441,Z 400.258,A -85,B 0,C 180,E1 -17830.48,E2 -17830.48} C_VEL
LIN {X 0,Y 270.402,Z 400.303,A -85,B 0,C 180,E1 -17835.064,E2 -17835.064} C_VEL
LIN {X 0,Y 270.299,Z 400.281,A -85,B 0,C 180,E1 -17839.755,E2 -17839.755} C_VEL
LIN {X 0,Y 270.272,Z 400.316,A -85,B 0,C 180,E1 -17844.585,E2 -17844.585} C_VEL
LIN {X 0,Y 270.267,Z 400.291,A -85,B 0,C 180,E1 -17847.908,E2 -17847.908} C_VEL
LIN {X 0,Y 270.181,Z 400.333,A -85,B 0,C 180,E1 -17851.347,E2 -17851.347} C_VEL
LIN {X 0,Y 270.212,Z 400.302,A -85,B 0,C 180,E1 -17854.903,E2 -17854.903} C_VEL
LIN {X 0,Y 270.22,Z 400.324,A -85,B 0,C 180,E1 -17858.716,E2 -17858.716} C_VEL
LIN {X 0,Y 270.169,Z 400.333,A -85,B 0,C 180,E1 -17863.25,E2 -17863.25} C_VEL
LIN {X 0,Y 270.172,Z 400.274,A -85,B 0,C 180,E1 -17867.442,E2 -17867.442} C_VEL
LIN {X 0,Y 270.211,Z 400.323,A -85,B 0,C 180,E1 -17871.375,E2 -17871.375} C_VEL
LIN {X 0,Y 270.213,Z 400.289,A -85,B 0,C 180,E1 -17875.096,E2 -17875.096} C_VEL
LIN {X 0,Y 270.249,Z 400.544,A -85,B 0,C 180,E1 -17879.292,E2 -17879.292} C_VEL
LIN {X 0,Y 270.532,Z 401.663,A -85,B 0,C 180,E1 -17879.534,E2 -17879.534} C_VEL
LIN {X 0,Y 282.954,Z 424.51,A -85,B 0,C 180,E1 -17881.676,E2 -17881.676} C_VEL
LIN {X 0,Y 291.275,Z 436.217,A -85,B 0,C 180,E1 -17882.88,E2 -17882.88} C_VEL
LIN {X 0,Y 303.657,Z 449.867,A -85,B 0,C 180,E1 -17884.448,E2 -17884.448} C_VEL
LIN {X 0,Y 312.724,Z 458.796,A -85,B 0,C 180,E1 -17885.696,E2 -17885.696} C_VEL
LIN {X 0,Y 321.117,Z 466.541,A -85,B 0,C 180,E1 -17887.032,E2 -17887.032} C_VEL
LIN {X 0,Y 329.658,Z 474.214,A -85,B 0,C 180,E1 -17888.614,E2 -17888.614} C_VEL
LIN {X 0,Y 338.439,Z 481.614,A -85,B 0,C 180,E1 -17890.442,E2 -17890.442} C_VEL
LIN {X 0,Y 343.868,Z 485.894,A -85,B 0,C 180,E1 -17891.683,E2 -17891.683} C_VEL
LIN {X 0,Y 350.159,Z 490.859,A -85,B 0,C 180,E1 -17893.244,E2 -17893.244} C_VEL
LIN {X 0,Y 354.981,Z 494.382,A -85,B 0,C 180,E1 -17894.557,E2 -17894.557} C_VEL
LIN {X 0,Y 360.935,Z 498.928,A -85,B 0,C 180,E1 -17896.381,E2 -17896.381} C_VEL
LIN {X 0,Y 365.944,Z 501.944,A -85,B 0,C 180,E1 -17898.117,E2 -17898.117} C_VEL
LIN {X 0,Y 369.111,Z 504.398,A -85,B 0,C 180,E1 -17899.391,E2 -17899.391} C_VEL
LIN {X 0,Y 372.81,Z 507.228,A -85,B 0,C 180,E1 -17901.128,E2 -17901.128} C_VEL
LIN {X 0,Y 376.103,Z 509.219,A -85,B 0,C 180,E1 -17903.005,E2 -17903.005} C_VEL
LIN {X 0,Y 378.71,Z 510.505,A -85,B 0,C 180,E1 -17904.946,E2 -17904.946} C_VEL
LIN {X 0,Y 380.674,Z 511.126,A -85,B 0,C 180,E1 -17907.083,E2 -17907.083} C_VEL
LIN {X 0,Y 381.48,Z 511.643,A -85,B 0,C 180,E1 -17908.944,E2 -17908.944} C_VEL
LIN {X 0,Y 381.623,Z 511.578,A -85,B 0,C 180,E1 -17910,E2 -17910} C_VEL
LIN {X 0,Y 381.313,Z 511.522,A -85,B 0,C 180,E1 -17911.584,E2 -17911.584} C_VEL
LIN {X 0,Y 380.222,Z 510.958,A -85,B 0,C 180,E1 -17913.515,E2 -17913.515} C_VEL
LIN {X 0,Y 378.396,Z 510.349,A -85,B 0,C 180,E1 -17915.328,E2 -17915.328} C_VEL
LIN {X 0,Y 375.789,Z 509.055,A -85,B 0,C 180,E1 -17917.2,E2 -17917.2} C_VEL
LIN {X 0,Y 372.377,Z 506.924,A -85,B 0,C 180,E1 -17919.095,E2 -17919.095} C_VEL
LIN {X 0,Y 368.692,Z 504.068,A -85,B 0,C 180,E1 -17920.785,E2 -17920.785} C_VEL
LIN {X 0,Y 366.164,Z 502.057,A -85,B 0,C 180,E1 -17921.803,E2 -17921.803} C_VEL
LIN {X 0,Y 361.297,Z 499.194,A -85,B 0,C 180,E1 -17923.498,E2 -17923.498} C_VEL
LIN {X 0,Y 355.428,Z 494.728,A -85,B 0,C 180,E1 -17925.318,E2 -17925.318} C_VEL
LIN {X 0,Y 350.866,Z 491.342,A -85,B 0,C 180,E1 -17926.574,E2 -17926.574} C_VEL
LIN {X 0,Y 344.78,Z 486.678,A -85,B 0,C 180,E1 -17928.099,E2 -17928.099} C_VEL
LIN {X 0,Y 340.444,Z 483.127,A -85,B 0,C 180,E1 -17929.112,E2 -17929.112} C_VEL
LIN {X 0,Y 334.027,Z 477.925,A -85,B 0,C 180,E1 -17930.497,E2 -17930.497} C_VEL
LIN {X 0,Y 325.947,Z 471.028,A -85,B 0,C 180,E1 -17932.083,E2 -17932.083} C_VEL
LIN {X 0,Y 317.977,Z 463.733,A -85,B 0,C 180,E1 -17933.487,E2 -17933.487} C_VEL
LIN {X 0,Y 309.038,Z 455.231,A -85,B 0,C 180,E1 -17934.836,E2 -17934.836} C_VEL
LIN {X 0,Y 300.829,Z 446.841,A -85,B 0,C 180,E1 -17935.907,E2 -17935.907} C_VEL
LIN {X 0,Y 290.792,Z 435.585,A -85,B 0,C 180,E1 -17937.186,E2 -17937.186} C_VEL
LIN {X 0,Y 282.832,Z 424.311,A -85,B 0,C 180,E1 -17938.343,E2 -17938.343} C_VEL
LIN {X 0,Y 276.509,Z 412.789,A -85,B 0,C 180,E1 -17939.395,E2 -17939.395} C_VEL
LIN {X 0,Y 271.443,Z 403.504,A -85,B 0,C 180,E1 -17940.282,E2 -17940.282} C_VEL
LIN {X 0,Y 270.368,Z 401.036,A -85,B 0,C 180,E1 -17940.562,E2 -17940.562} C_VEL
LIN {X 0,Y 270.202,Z 400.376,A -85,B 0,C 180,E1 -17940.872,E2 -17940.872} C_VEL
LIN {X 0,Y 270.21,Z 400.289,A -85,B 0,C 180,E1 -17944.903,E2 -17944.903} C_VEL
LIN {X 0,Y 270.217,Z 400.321,A -85,B 0,C 180,E1 -17948.717,E2 -17948.717} C_VEL
LIN {X 0,Y 270.166,Z 400.281,A -85,B 0,C 180,E1 -17953.25,E2 -17953.25} C_VEL
LIN {X 0,Y 270.189,Z 400.326,A -85,B 0,C 180,E1 -17957.446,E2 -17957.446} C_VEL
LIN {X 0,Y 270.239,Z 400.323,A -85,B 0,C 180,E1 -17961.381,E2 -17961.381} C_VEL
LIN {X 0,Y 270.21,Z 400.303,A -85,B 0,C 180,E1 -17965.097,E2 -17965.097} C_VEL
LIN {X 0,Y 270.194,Z 400.329,A -85,B 0,C 180,E1 -17969.131,E2 -17969.131} C_VEL
LIN {X 0,Y 270.259,Z 400.292,A -85,B 0,C 180,E1 -17972.146,E2 -17972.146} C_VEL
LIN {X 0,Y 270.271,Z 400.316,A -85,B 0,C 180,E1 -17975.52,E2 -17975.52} C_VEL
LIN {X 0,Y 270.296,Z 400.281,A -85,B 0,C 180,E1 -17980.245,E2 -17980.245} C_VEL
LIN {X 0,Y 270.398,Z 400.303,A -85,B 0,C 180,E1 -17984.936,E2 -17984.936} C_VEL
LIN {X 0,Y 270.437,Z 400.258,A -85,B 0,C 180,E1 -17989.52,E2 -17989.52} C_VEL
LIN {X 0,Y 270.606,Z 400.262,A -85,B 0,C 180,E1 -17992.54,E2 -17992.54} C_VEL
LIN {X 0,Y 270.783,Z 400.217,A -85,B 0,C 180,E1 -17998.514,E2 -17998.514} C_VEL
LIN {X 0,Y 270.783,Z 400.229,A -85,B 0,C 180,E1 -18001.488,E2 -18001.488} C_VEL
LIN {X 0,Y 270.607,Z 400.251,A -85,B 0,C 180,E1 -18007.462,E2 -18007.462} C_VEL
LIN {X 0,Y 270.438,Z 400.26,A -85,B 0,C 180,E1 -18010.482,E2 -18010.482} C_VEL
LIN {X 0,Y 270.399,Z 400.296,A -85,B 0,C 180,E1 -18015.066,E2 -18015.066} C_VEL
LIN {X 0,Y 270.298,Z 400.285,A -85,B 0,C 180,E1 -18019.757,E2 -18019.757} C_VEL
LIN {X 0,Y 270.272,Z 400.306,A -85,B 0,C 180,E1 -18024.587,E2 -18024.587} C_VEL
LIN {X 0,Y 270.27,Z 400.295,A -85,B 0,C 180,E1 -18027.91,E2 -18027.91} C_VEL
LIN {X 0,Y 270.183,Z 400.329,A -85,B 0,C 180,E1 -18031.349,E2 -18031.349} C_VEL
LIN {X 0,Y 270.179,Z 400.311,A -85,B 0,C 180,E1 -18032.758,E2 -18032.758} C_VEL
LIN {X 0,Y 269.565,Z 400.388,A -85,B 0,C 180,E1 -18034.003,E2 -18034.003} C_VEL
LIN {X 0,Y 266.728,Z 400.753,A -85,B 0,C 180,E1 -18036.032,E2 -18036.032} C_VEL
LIN {X 0,Y 264.288,Z 401.065,A -85,B 0,C 180,E1 -18037.681,E2 -18037.681} C_VEL
LIN {X 0,Y 263.239,Z 401.183,A -85,B 0,C 180,E1 -18038.961,E2 -18038.961} C_VEL
LIN {X 0,Y 263.154,Z 401.19,A -85,B 0,C 180,E1 -18039.394,E2 -18039.394} C_VEL
LIN {X 0,Y 263.206,Z 401.198,A -85,B 0,C 180,E1 -18041.878,E2 -18041.878} C_VEL
LIN {X 0,Y 263.138,Z 401.211,A -85,B 0,C 180,E1 -18046.149,E2 -18046.149} C_VEL
LIN {X 0,Y 263.107,Z 401.182,A -85,B 0,C 180,E1 -18050.129,E2 -18050.129} C_VEL
LIN {X 0,Y 263.214,Z 401.404,A -85,B 0,C 180,E1 -18051.637,E2 -18051.637} C_VEL
LIN {X 0,Y 264.803,Z 408.725,A -85,B 0,C 180,E1 -18055.363,E2 -18055.363} C_VEL
LIN {X 0,Y 266.359,Z 416.344,A -85,B 0,C 180,E1 -18058.994,E2 -18058.994} C_VEL
LIN {X 0,Y 267.885,Z 419.986,A -85,B 0,C 180,E1 -18059.385,E2 -18059.385} C_VEL
LIN {X 0,Y 272.797,Z 432.144,A -85,B 0,C 180,E1 -18060.35,E2 -18060.35} C_VEL
LIN {X 0,Y 277.6,Z 456.623,A -85,B 0,C 180,E1 -18061.615,E2 -18061.615} C_VEL
LIN {X 0,Y 279.226,Z 466.909,A -85,B 0,C 180,E1 -18062.086,E2 -18062.086} C_VEL
LIN {X 0,Y 277.485,Z 521.498,A -85,B 0,C 180,E1 -18063.488,E2 -18063.488} C_VEL
LIN {X 0,Y 276.784,Z 532.177,A -85,B 0,C 180,E1 -18063.923,E2 -18063.923} C_VEL
LIN {X 0,Y 275.695,Z 542.56,A -85,B 0,C 180,E1 -18064.522,E2 -18064.522} C_VEL
LIN {X 0,Y 274.557,Z 551.651,A -85,B 0,C 180,E1 -18065.219,E2 -18065.219} C_VEL
LIN {X 0,Y 273.283,Z 560.796,A -85,B 0,C 180,E1 -18066.107,E2 -18066.107} C_VEL
LIN {X 0,Y 271.71,Z 569.793,A -85,B 0,C 180,E1 -18067.172,E2 -18067.172} C_VEL
LIN {X 0,Y 270.081,Z 578.517,A -85,B 0,C 180,E1 -18068.436,E2 -18068.436} C_VEL
LIN {X 0,Y 268.598,Z 585.937,A -85,B 0,C 180,E1 -18069.716,E2 -18069.716} C_VEL
LIN {X 0,Y 266.864,Z 594.734,A -85,B 0,C 180,E1 -18071.578,E2 -18071.578} C_VEL
LIN {X 0,Y 265.594,Z 600.724,A -85,B 0,C 180,E1 -18073.078,E2 -18073.078} C_VEL
LIN {X 0,Y 264.244,Z 607.035,A -85,B 0,C 180,E1 -18074.971,E2 -18074.971} C_VEL
LIN {X 0,Y 263.086,Z 612.308,A -85,B 0,C 180,E1 -18076.876,E2 -18076.876} C_VEL
LIN {X 0,Y 262.135,Z 617.404,A -85,B 0,C 180,E1 -18079.184,E2 -18079.184} C_VEL
LIN {X 0,Y 261.517,Z 621.372,A -85,B 0,C 180,E1 -18081.501,E2 -18081.501} C_VEL
LIN {X 0,Y 261.087,Z 625.346,A -85,B 0,C 180,E1 -18084.865,E2 -18084.865} C_VEL
LIN {X 0,Y 261.055,Z 626.743,A -85,B 0,C 180,E1 -18086.914,E2 -18086.914} C_VEL
LIN {X 0,Y 261.118,Z 627.621,A -85,B 0,C 180,E1 -18090,E2 -18090} C_VEL
LIN {X 0,Y 261.053,Z 626.742,A -85,B 0,C 180,E1 -18093.087,E2 -18093.087} C_VEL
LIN {X 0,Y 261.088,Z 625.343,A -85,B 0,C 180,E1 -18095.138,E2 -18095.138} C_VEL
LIN {X 0,Y 261.517,Z 621.37,A -85,B 0,C 180,E1 -18098.5,E2 -18098.5} C_VEL
LIN {X 0,Y 262.136,Z 617.403,A -85,B 0,C 180,E1 -18100.817,E2 -18100.817} C_VEL
LIN {X 0,Y 263.084,Z 612.306,A -85,B 0,C 180,E1 -18103.125,E2 -18103.125} C_VEL
LIN {X 0,Y 264.81,Z 604.658,A -85,B 0,C 180,E1 -18105.786,E2 -18105.786} C_VEL
LIN {X 0,Y 266.291,Z 597.855,A -85,B 0,C 180,E1 -18107.669,E2 -18107.669} C_VEL
LIN {X 0,Y 267.887,Z 589.636,A -85,B 0,C 180,E1 -18109.542,E2 -18109.542} C_VEL
LIN {X 0,Y 269.454,Z 581.807,A -85,B 0,C 180,E1 -18111.016,E2 -18111.016} C_VEL
LIN {X 0,Y 271.029,Z 573.726,A -85,B 0,C 180,E1 -18112.287,E2 -18112.287} C_VEL
LIN {X 0,Y 272.741,Z 563.967,A -85,B 0,C 180,E1 -18113.541,E2 -18113.541} C_VEL
LIN {X 0,Y 274.027,Z 555.578,A -85,B 0,C 180,E1 -18114.429,E2 -18114.429} C_VEL
LIN {X 0,Y 275.379,Z 545.072,A -85,B 0,C 180,E1 -18115.308,E2 -18115.308} C_VEL
LIN {X 0,Y 276.527,Z 534.742,A -85,B 0,C 180,E1 -18115.952,E2 -18115.952} C_VEL
LIN {X 0,Y 277.403,Z 524.022,A -85,B 0,C 180,E1 -18116.42,E2 -18116.42} C_VEL
LIN {X 0,Y 278.171,Z 499.894,A -85,B 0,C 180,E1 -18117.088,E2 -18117.088} C_VEL
LIN {X 0,Y 279.106,Z 465.849,A -85,B 0,C 180,E1 -18117.957,E2 -18117.957} C_VEL
LIN {X 0,Y 275.193,Z 443.808,A -85,B 0,C 180,E1 -18119.028,E2 -18119.028} C_VEL
LIN {X 0,Y 272.268,Z 430.465,A -85,B 0,C 180,E1 -18119.763,E2 -18119.763} C_VEL
LIN {X 0,Y 266.43,Z 416.725,A -85,B 0,C 180,E1 -18120.934,E2 -18120.934} C_VEL
LIN {X 0,Y 266.152,Z 415.574,A -85,B 0,C 180,E1 -18121.294,E2 -18121.294} C_VEL
LIN {X 0,Y 264.619,Z 407.784,A -85,B 0,C 180,E1 -18125.101,E2 -18125.101} C_VEL
LIN {X 0,Y 263.202,Z 401.288,A -85,B 0,C 180,E1 -18128.486,E2 -18128.486} C_VEL
LIN {X 0,Y 263.134,Z 401.182,A -85,B 0,C 180,E1 -18131.891,E2 -18131.891} C_VEL
LIN {X 0,Y 263.15,Z 401.196,A -85,B 0,C 180,E1 -18136.145,E2 -18136.145} C_VEL
LIN {X 0,Y 263.213,Z 401.196,A -85,B 0,C 180,E1 -18138.385,E2 -18138.385} C_VEL
LIN {X 0,Y 263.209,Z 401.199,A -85,B 0,C 180,E1 -18143.229,E2 -18143.229} C_VEL
LIN {X 0,Y 263.186,Z 401.177,A -85,B 0,C 180,E1 -18145.89,E2 -18145.89} C_VEL
LIN {X 0,Y 263.153,Z 401.206,A -85,B 0,C 180,E1 -18149.506,E2 -18149.506} C_VEL
LIN {X 0,Y 263.194,Z 401.168,A -85,B 0,C 180,E1 -18153.002,E2 -18153.002} C_VEL
LIN {X 0,Y 263.186,Z 401.199,A -85,B 0,C 180,E1 -18156.386,E2 -18156.386} C_VEL
LIN {X 0,Y 263.264,Z 401.168,A -85,B 0,C 180,E1 -18159.693,E2 -18159.693} C_VEL
LIN {X 0,Y 263.351,Z 401.172,A -85,B 0,C 180,E1 -18164.521,E2 -18164.521} C_VEL
LIN {X 0,Y 263.374,Z 401.141,A -85,B 0,C 180,E1 -18169.234,E2 -18169.234} C_VEL
LIN {X 0,Y 263.573,Z 401.122,A -85,B 0,C 180,E1 -18172.338,E2 -18172.338} C_VEL
LIN {X 0,Y 263.751,Z 401.105,A -85,B 0,C 180,E1 -18178.472,E2 -18178.472} C_VEL
LIN {X 0,Y 263.75,Z 401.093,A -85,B 0,C 180,E1 -18181.526,E2 -18181.526} C_VEL
LIN {X 0,Y 263.571,Z 401.136,A -85,B 0,C 180,E1 -18187.661,E2 -18187.661} C_VEL
LIN {X 0,Y 263.373,Z 401.139,A -85,B 0,C 180,E1 -18190.765,E2 -18190.765} C_VEL
LIN {X 0,Y 263.35,Z 401.18,A -85,B 0,C 180,E1 -18195.477,E2 -18195.477} C_VEL
LIN {X 0,Y 263.262,Z 401.161,A -85,B 0,C 180,E1 -18200.306,E2 -18200.306} C_VEL
LIN {X 0,Y 263.206,Z 401.187,A -85,B 0,C 180,E1 -18205.291,E2 -18205.291} C_VEL
LIN {X 0,Y 263.163,Z 401.183,A -85,B 0,C 180,E1 -18208.73,E2 -18208.73} C_VEL
LIN {X 0,Y 263.131,Z 401.206,A -85,B 0,C 180,E1 -18212.287,E2 -18212.287} C_VEL
LIN {X 0,Y 263.185,Z 401.186,A -85,B 0,C 180,E1 -18215.977,E2 -18215.977} C_VEL
LIN {X 0,Y 263.111,Z 401.195,A -85,B 0,C 180,E1 -18219.87,E2 -18219.87} C_VEL
LIN {X 0,Y 263.125,Z 401.207,A -85,B 0,C 180,E1 -18223.982,E2 -18223.982} C_VEL
LIN {X 0,Y 263.123,Z 401.15,A -85,B 0,C 180,E1 -18228.405,E2 -18228.405} C_VEL
LIN {X 0,Y 263.168,Z 401.206,A -85,B 0,C 180,E1 -18232.104,E2 -18232.104} C_VEL
LIN {X 0,Y 263.181,Z 401.165,A -85,B 0,C 180,E1 -18235.89,E2 -18235.89} C_VEL
LIN {X 0,Y 263.171,Z 401.411,A -85,B 0,C 180,E1 -18238.396,E2 -18238.396} C_VEL
LIN {X 0,Y 263.401,Z 402.392,A -85,B 0,C 180,E1 -18238.627,E2 -18238.627} C_VEL
LIN {X 0,Y 271.565,Z 417.526,A -85,B 0,C 180,E1 -18240.153,E2 -18240.153} C_VEL
LIN {X 0,Y 277.977,Z 429.124,A -85,B 0,C 180,E1 -18241.251,E2 -18241.251} C_VEL
LIN {X 0,Y 286.377,Z 440.985,A -85,B 0,C 180,E1 -18242.505,E2 -18242.505} C_VEL
LIN {X 0,Y 298.221,Z 454.181,A -85,B 0,C 180,E1 -18244.04,E2 -18244.04} C_VEL
LIN {X 0,Y 308.382,Z 464.095,A -85,B 0,C 180,E1 -18245.331,E2 -18245.331} C_VEL
LIN {X 0,Y 316.967,Z 471.927,A -85,B 0,C 180,E1 -18246.611,E2 -18246.611} C_VEL
LIN {X 0,Y 324.916,Z 478.937,A -85,B 0,C 180,E1 -18247.98,E2 -18247.98} C_VEL
LIN {X 0,Y 332.474,Z 485.274,A -85,B 0,C 180,E1 -18249.445,E2 -18249.445} C_VEL
LIN {X 0,Y 339.23,Z 490.461,A -85,B 0,C 180,E1 -18250.88,E2 -18250.88} C_VEL
LIN {X 0,Y 346.455,Z 496.313,A -85,B 0,C 180,E1 -18252.585,E2 -18252.585} C_VEL
LIN {X 0,Y 352.586,Z 500.686,A -85,B 0,C 180,E1 -18254.193,E2 -18254.193} C_VEL
LIN {X 0,Y 358.005,Z 504.875,A -85,B 0,C 180,E1 -18255.788,E2 -18255.788} C_VEL
LIN {X 0,Y 363.273,Z 508.166,A -85,B 0,C 180,E1 -18257.503,E2 -18257.503} C_VEL
LIN {X 0,Y 366.2,Z 509.949,A -85,B 0,C 180,E1 -18258.577,E2 -18258.577} C_VEL
LIN {X 0,Y 370.364,Z 513.309,A -85,B 0,C 180,E1 -18260.389,E2 -18260.389} C_VEL
LIN {X 0,Y 373.747,Z 515.486,A -85,B 0,C 180,E1 -18262.13,E2 -18262.13} C_VEL
LIN {X 0,Y 376.72,Z 517.043,A -85,B 0,C 180,E1 -18264.046,E2 -18264.046} C_VEL
LIN {X 0,Y 378.685,Z 517.811,A -85,B 0,C 180,E1 -18265.742,E2 -18265.742} C_VEL
LIN {X 0,Y 379.929,Z 518.267,A -85,B 0,C 180,E1 -18267.3,E2 -18267.3} C_VEL
LIN {X 0,Y 380.613,Z 518.689,A -85,B 0,C 180,E1 -18268.942,E2 -18268.942} C_VEL
LIN {X 0,Y 380.758,Z 518.624,A -85,B 0,C 180,E1 -18270,E2 -18270} C_VEL
LIN {X 0,Y 380.444,Z 518.568,A -85,B 0,C 180,E1 -18271.588,E2 -18271.588} C_VEL
LIN {X 0,Y 379.6,Z 518.064,A -85,B 0,C 180,E1 -18273.184,E2 -18273.184} C_VEL
LIN {X 0,Y 377.82,Z 517.538,A -85,B 0,C 180,E1 -18275.065,E2 -18275.065} C_VEL
LIN {X 0,Y 375.25,Z 516.304,A -85,B 0,C 180,E1 -18276.967,E2 -18276.967} C_VEL
LIN {X 0,Y 371.736,Z 514.246,A -85,B 0,C 180,E1 -18278.954,E2 -18278.954} C_VEL
LIN {X 0,Y 367.897,Z 511.434,A -85,B 0,C 180,E1 -18280.718,E2 -18280.718} C_VEL
LIN {X 0,Y 364.634,Z 508.868,A -85,B 0,C 180,E1 -18282.013,E2 -18282.013} C_VEL
LIN {X 0,Y 359.517,Z 505.875,A -85,B 0,C 180,E1 -18283.755,E2 -18283.755} C_VEL
LIN {X 0,Y 353.672,Z 501.563,A -85,B 0,C 180,E1 -18285.504,E2 -18285.504} C_VEL
LIN {X 0,Y 349.563,Z 498.472,A -85,B 0,C 180,E1 -18286.629,E2 -18286.629} C_VEL
LIN {X 0,Y 342.943,Z 493.605,A -85,B 0,C 180,E1 -18288.257,E2 -18288.257} C_VEL
LIN {X 0,Y 337.19,Z 488.978,A -85,B 0,C 180,E1 -18289.567,E2 -18289.567} C_VEL
LIN {X 0,Y 330.045,Z 483.153,A -85,B 0,C 180,E1 -18291.051,E2 -18291.051} C_VEL
LIN {X 0,Y 321.397,Z 475.839,A -85,B 0,C 180,E1 -18292.659,E2 -18292.659} C_VEL
LIN {X 0,Y 312.817,Z 468.165,A -85,B 0,C 180,E1 -18294.036,E2 -18294.036} C_VEL
LIN {X 0,Y 303.948,Z 459.84,A -85,B 0,C 180,E1 -18295.259,E2 -18295.259} C_VEL
LIN {X 0,Y 291.377,Z 446.852,A -85,B 0,C 180,E1 -18296.821,E2 -18296.821} C_VEL
LIN {X 0,Y 284.094,Z 437.898,A -85,B 0,C 180,E1 -18297.823,E2 -18297.823} C_VEL
LIN {X 0,Y 277.257,Z 428.018,A -85,B 0,C 180,E1 -18298.864,E2 -18298.864} C_VEL
LIN {X 0,Y 264.624,Z 404.76,A -85,B 0,C 180,E1 -18301.116,E2 -18301.116} C_VEL
LIN {X 0,Y 263.299,Z 402.065,A -85,B 0,C 180,E1 -18301.427,E2 -18301.427} C_VEL
LIN {X 0,Y 263.124,Z 401.266,A -85,B 0,C 180,E1 -18301.786,E2 -18301.786} C_VEL
LIN {X 0,Y 263.168,Z 401.167,A -85,B 0,C 180,E1 -18304.122,E2 -18304.122} C_VEL
LIN {X 0,Y 263.165,Z 401.206,A -85,B 0,C 180,E1 -18307.895,E2 -18307.895} C_VEL
LIN {X 0,Y 263.12,Z 401.15,A -85,B 0,C 180,E1 -18311.893,E2 -18311.893} C_VEL
LIN {X 0,Y 263.13,Z 401.207,A -85,B 0,C 180,E1 -18316.148,E2 -18316.148} C_VEL
LIN {X 0,Y 263.133,Z 401.192,A -85,B 0,C 180,E1 -18320.134,E2 -18320.134} C_VEL
LIN {X 0,Y 263.184,Z 401.187,A -85,B 0,C 180,E1 -18324.023,E2 -18324.023} C_VEL
LIN {X 0,Y 263.127,Z 401.206,A -85,B 0,C 180,E1 -18327.712,E2 -18327.712} C_VEL
LIN {X 0,Y 263.195,Z 401.174,A -85,B 0,C 180,E1 -18331.784,E2 -18331.784} C_VEL
LIN {X 0,Y 263.22,Z 401.192,A -85,B 0,C 180,E1 -18335.201,E2 -18335.201} C_VEL
LIN {X 0,Y 263.258,Z 401.162,A -85,B 0,C 180,E1 -18339.694,E2 -18339.694} C_VEL
LIN {X 0,Y 263.345,Z 401.18,A -85,B 0,C 180,E1 -18344.523,E2 -18344.523} C_VEL
LIN {X 0,Y 263.369,Z 401.139,A -85,B 0,C 180,E1 -18349.235,E2 -18349.235} C_VEL
LIN {X 0,Y 263.567,Z 401.136,A -85,B 0,C 180,E1 -18352.339,E2 -18352.339} C_VEL
LIN {X 0,Y 263.747,Z 401.093,A -85,B 0,C 180,E1 -18358.474,E2 -18358.474} C_VEL
LIN {X 0,Y 263.747,Z 401.105,A -85,B 0,C 180,E1 -18361.528,E2 -18361.528} C_VEL
LIN {X 0,Y 263.569,Z 401.123,A -85,B 0,C 180,E1 -18367.663,E2 -18367.663} C_VEL
LIN {X 0,Y 263.37,Z 401.143,A -85,B 0,C 180,E1 -18370.767,E2 -18370.767} C_VEL
LIN {X 0,Y 263.347,Z 401.173,A -85,B 0,C 180,E1 -18375.479,E2 -18375.479} C_VEL
LIN {X 0,Y 263.261,Z 401.168,A -85,B 0,C 180,E1 -18380.308,E2 -18380.308} C_VEL
LIN {X 0,Y 263.206,Z 401.176,A -85,B 0,C 180,E1 -18385.292,E2 -18385.292} C_VEL
LIN {X 0,Y 263.178,Z 401.188,A -85,B 0,C 180,E1 -18388.731,E2 -18388.731} C_VEL
LIN {X 0,Y 263.12,Z 401.191,A -85,B 0,C 180,E1 -18392.755,E2 -18392.755} C_VEL
LIN {X 0,Y 263.205,Z 401.199,A -85,B 0,C 180,E1 -18396.772,E2 -18396.772} C_VEL
LIN {X 0,Y 263.154,Z 401.19,A -85,B 0,C 180,E1 -18399.394,E2 -18399.394} C_VEL
LIN {X 0,Y 262.482,Z 401.278,A -85,B 0,C 180,E1 -18400.672,E2 -18400.672} C_VEL
LIN {X 0,Y 259.607,Z 401.646,A -85,B 0,C 180,E1 -18402.753,E2 -18402.753} C_VEL
LIN {X 0,Y 257.173,Z 401.948,A -85,B 0,C 180,E1 -18404.447,E2 -18404.447} C_VEL
LIN {X 0,Y 256.139,Z 402.079,A -85,B 0,C 180,E1 -18405.76,E2 -18405.76} C_VEL
LIN {X 0,Y 256.06,Z 402.086,A -85,B 0,C 180,E1 -18406.205,E2 -18406.205} C_VEL
LIN {X 0,Y 256.118,Z 402.178,A -85,B 0,C 180,E1 -18410.868,E2 -18410.868} C_VEL
LIN {X 0,Y 257.504,Z 408.161,A -85,B 0,C 180,E1 -18414.072,E2 -18414.072} C_VEL
LIN {X 0,Y 259.089,Z 416.025,A -85,B 0,C 180,E1 -18417.997,E2 -18417.997} C_VEL
LIN {X 0,Y 259.81,Z 418.195,A -85,B 0,C 180,E1 -18418.277,E2 -18418.277} C_VEL
LIN {X 0,Y 265.55,Z 431.119,A -85,B 0,C 180,E1 -18419.432,E2 -18419.432} C_VEL
LIN {X 0,Y 267.082,Z 435.643,A -85,B 0,C 180,E1 -18419.762,E2 -18419.762} C_VEL
LIN {X 0,Y 271.604,Z 459.16,A -85,B 0,C 180,E1 -18421.01,E2 -18421.01} C_VEL
LIN {X 0,Y 272.94,Z 467.59,A -85,B 0,C 180,E1 -18421.411,E2 -18421.411} C_VEL
LIN {X 0,Y 271.072,Z 522.667,A -85,B 0,C 180,E1 -18422.867,E2 -18422.867} C_VEL
LIN {X 0,Y 270.347,Z 532.878,A -85,B 0,C 180,E1 -18423.308,E2 -18423.308} C_VEL
LIN {X 0,Y 269.309,Z 542.365,A -85,B 0,C 180,E1 -18423.873,E2 -18423.873} C_VEL
LIN {X 0,Y 268.128,Z 551.456,A -85,B 0,C 180,E1 -18424.583,E2 -18424.583} C_VEL
LIN {X 0,Y 266.771,Z 560.6,A -85,B 0,C 180,E1 -18425.486,E2 -18425.486} C_VEL
LIN {X 0,Y 265.178,Z 569.598,A -85,B 0,C 180,E1 -18426.576,E2 -18426.576} C_VEL
LIN {X 0,Y 263.483,Z 578.322,A -85,B 0,C 180,E1 -18427.868,E2 -18427.868} C_VEL
LIN {X 0,Y 261.945,Z 585.741,A -85,B 0,C 180,E1 -18429.177,E2 -18429.177} C_VEL
LIN {X 0,Y 260.09,Z 594.395,A -85,B 0,C 180,E1 -18431.043,E2 -18431.043} C_VEL
LIN {X 0,Y 258.798,Z 600.529,A -85,B 0,C 180,E1 -18432.62,E2 -18432.62} C_VEL
LIN {X 0,Y 257.384,Z 606.84,A -85,B 0,C 180,E1 -18434.561,E2 -18434.561} C_VEL
LIN {X 0,Y 256.163,Z 612.113,A -85,B 0,C 180,E1 -18436.515,E2 -18436.515} C_VEL
LIN {X 0,Y 255.128,Z 617.208,A -85,B 0,C 180,E1 -18438.883,E2 -18438.883} C_VEL
LIN {X 0,Y 254.473,Z 621.176,A -85,B 0,C 180,E1 -18441.264,E2 -18441.264} C_VEL
LIN {X 0,Y 254.068,Z 624.113,A -85,B 0,C 180,E1 -18443.648,E2 -18443.648} C_VEL
LIN {X 0,Y 253.976,Z 625.617,A -85,B 0,C 180,E1 -18445.239,E2 -18445.239} C_VEL
LIN {X 0,Y 253.996,Z 627.146,A -85,B 0,C 180,E1 -18448.415,E2 -18448.415} C_VEL
LIN {X 0,Y 254.046,Z 627.427,A -85,B 0,C 180,E1 -18450,E2 -18450} C_VEL
LIN {X 0,Y 253.952,Z 626.547,A -85,B 0,C 180,E1 -18453.173,E2 -18453.173} C_VEL
LIN {X 0,Y 253.993,Z 625.382,A -85,B 0,C 180,E1 -18455.039,E2 -18455.039} C_VEL
LIN {X 0,Y 254.305,Z 622.264,A -85,B 0,C 180,E1 -18457.943,E2 -18457.943} C_VEL
LIN {X 0,Y 254.863,Z 618.635,A -85,B 0,C 180,E1 -18460.326,E2 -18460.326} C_VEL
LIN {X 0,Y 255.732,Z 613.9,A -85,B 0,C 180,E1 -18462.701,E2 -18462.701} C_VEL
LIN {X 0,Y 257.089,Z 607.929,A -85,B 0,C 180,E1 -18465.053,E2 -18465.053} C_VEL
LIN {X 0,Y 258.173,Z 603.149,A -85,B 0,C 180,E1 -18466.609,E2 -18466.609} C_VEL
LIN {X 0,Y 259.725,Z 596.579,A -85,B 0,C 180,E1 -18468.413,E2 -18468.413} C_VEL
LIN {X 0,Y 261.173,Z 589.44,A -85,B 0,C 180,E1 -18470.065,E2 -18470.065} C_VEL
LIN {X 0,Y 262.831,Z 581.612,A -85,B 0,C 180,E1 -18471.572,E2 -18471.572} C_VEL
LIN {X 0,Y 264.462,Z 573.53,A -85,B 0,C 180,E1 -18472.871,E2 -18472.871} C_VEL
LIN {X 0,Y 266.23,Z 563.771,A -85,B 0,C 180,E1 -18474.153,E2 -18474.153} C_VEL
LIN {X 0,Y 267.563,Z 555.382,A -85,B 0,C 180,E1 -18475.059,E2 -18475.059} C_VEL
LIN {X 0,Y 268.984,Z 544.877,A -85,B 0,C 180,E1 -18475.954,E2 -18475.954} C_VEL
LIN {X 0,Y 270.166,Z 534.57,A -85,B 0,C 180,E1 -18476.609,E2 -18476.609} C_VEL
LIN {X 0,Y 271.067,Z 523.918,A -85,B 0,C 180,E1 -18477.084,E2 -18477.084} C_VEL
LIN {X 0,Y 271.83,Z 501.045,A -85,B 0,C 180,E1 -18477.735,E2 -18477.735} C_VEL
LIN {X 0,Y 272.871,Z 466.942,A -85,B 0,C 180,E1 -18478.616,E2 -18478.616} C_VEL
LIN {X 0,Y 268.925,Z 444.707,A -85,B 0,C 180,E1 -18479.738,E2 -18479.738} C_VEL
LIN {X 0,Y 266.41,Z 433.267,A -85,B 0,C 180,E1 -18480.394,E2 -18480.394} C_VEL
LIN {X 0,Y 260.335,Z 419.37,A -85,B 0,C 180,E1 -18481.615,E2 -18481.615} C_VEL
LIN {X 0,Y 259.113,Z 416.183,A -85,B 0,C 180,E1 -18481.955,E2 -18481.955} C_VEL
LIN {X 0,Y 257.791,Z 409.726,A -85,B 0,C 180,E1 -18485.126,E2 -18485.126} C_VEL
LIN {X 0,Y 256.545,Z 403.915,A -85,B 0,C 180,E1 -18488.166,E2 -18488.166} C_VEL
LIN {X 0,Y 256.111,Z 402.134,A -85,B 0,C 180,E1 -18489.293,E2 -18489.293} C_VEL
LIN {X 0,Y 256.075,Z 402.085,A -85,B 0,C 180,E1 -18493.324,E2 -18493.324} C_VEL
LIN {X 0,Y 256.157,Z 402.079,A -85,B 0,C 180,E1 -18497.798,E2 -18497.798} C_VEL
LIN {X 0,Y 256.112,Z 402.069,A -85,B 0,C 180,E1 -18500.864,E2 -18500.864} C_VEL
LIN {X 0,Y 256.124,Z 402.063,A -85,B 0,C 180,E1 -18504.813,E2 -18504.813} C_VEL
LIN {X 0,Y 256.095,Z 402.083,A -85,B 0,C 180,E1 -18508.572,E2 -18508.572} C_VEL
LIN {X 0,Y 256.143,Z 402.051,A -85,B 0,C 180,E1 -18512.195,E2 -18512.195} C_VEL
LIN {X 0,Y 256.169,Z 402.064,A -85,B 0,C 180,E1 -18515.698,E2 -18515.698} C_VEL
LIN {X 0,Y 256.168,Z 402.059,A -85,B 0,C 180,E1 -18519.104,E2 -18519.104} C_VEL
LIN {X 0,Y 256.3,Z 402.043,A -85,B 0,C 180,E1 -18524.084,E2 -18524.084} C_VEL
LIN {X 0,Y 256.31,Z 402.024,A -85,B 0,C 180,E1 -18528.933,E2 -18528.933} C_VEL
LIN {X 0,Y 256.541,Z 401.993,A -85,B 0,C 180,E1 -18532.126,E2 -18532.126} C_VEL
LIN {X 0,Y 256.714,Z 401.98,A -85,B 0,C 180,E1 -18538.43,E2 -18538.43} C_VEL
LIN {X 0,Y 256.713,Z 401.969,A -85,B 0,C 180,E1 -18541.568,E2 -18541.568} C_VEL
LIN {X 0,Y 256.539,Z 402.01,A -85,B 0,C 180,E1 -18547.872,E2 -18547.872} C_VEL
LIN {X 0,Y 256.309,Z 402.02,A -85,B 0,C 180,E1 -18551.065,E2 -18551.065} C_VEL
LIN {X 0,Y 256.299,Z 402.054,A -85,B 0,C 180,E1 -18555.914,E2 -18555.914} C_VEL
LIN {X 0,Y 256.165,Z 402.052,A -85,B 0,C 180,E1 -18560.894,E2 -18560.894} C_VEL
LIN {X 0,Y 256.186,Z 402.063,A -85,B 0,C 180,E1 -18565.138,E2 -18565.138} C_VEL
LIN {X 0,Y 256.101,Z 402.073,A -85,B 0,C 180,E1 -18569.6,E2 -18569.6} C_VEL
LIN {X 0,Y 256.083,Z 402.069,A -85,B 0,C 180,E1 -18573.289,E2 -18573.289} C_VEL
LIN {X 0,Y 256.126,Z 402.081,A -85,B 0,C 180,E1 -18577.274,E2 -18577.274} C_VEL
LIN {X 0,Y 256.054,Z 402.071,A -85,B 0,C 180,E1 -18581.202,E2 -18581.202} C_VEL
LIN {X 0,Y 256.059,Z 402.057,A -85,B 0,C 180,E1 -18585.528,E2 -18585.528} C_VEL
LIN {X 0,Y 256.055,Z 402.032,A -85,B 0,C 180,E1 -18588.797,E2 -18588.797} C_VEL
LIN {X 0,Y 256.146,Z 402.069,A -85,B 0,C 180,E1 -18592.87,E2 -18592.87} C_VEL
LIN {X 0,Y 256.098,Z 402.11,A -85,B 0,C 180,E1 -18597.302,E2 -18597.302} C_VEL
LIN {X 0,Y 256.254,Z 402.973,A -85,B 0,C 180,E1 -18597.642,E2 -18597.642} C_VEL
LIN {X 0,Y 257.774,Z 405.854,A -85,B 0,C 180,E1 -18597.988,E2 -18597.988} C_VEL
LIN {X 0,Y 266.206,Z 421.399,A -85,B 0,C 180,E1 -18599.603,E2 -18599.603} C_VEL
LIN {X 0,Y 272.708,Z 433.264,A -85,B 0,C 180,E1 -18600.759,E2 -18600.759} C_VEL
LIN {X 0,Y 281.191,Z 445.367,A -85,B 0,C 180,E1 -18602.074,E2 -18602.074} C_VEL
LIN {X 0,Y 291.254,Z 456.761,A -85,B 0,C 180,E1 -18603.435,E2 -18603.435} C_VEL
LIN {X 0,Y 303.289,Z 468.804,A -85,B 0,C 180,E1 -18604.918,E2 -18604.918} C_VEL
LIN {X 0,Y 312.133,Z 476.74,A -85,B 0,C 180,E1 -18606.121,E2 -18606.121} C_VEL
LIN {X 0,Y 321.003,Z 484.407,A -85,B 0,C 180,E1 -18607.53,E2 -18607.53} C_VEL
LIN {X 0,Y 329.966,Z 491.794,A -85,B 0,C 180,E1 -18609.196,E2 -18609.196} C_VEL
LIN {X 0,Y 338.628,Z 498.447,A -85,B 0,C 180,E1 -18611.015,E2 -18611.015} C_VEL
LIN {X 0,Y 345.61,Z 503.814,A -85,B 0,C 180,E1 -18612.652,E2 -18612.652} C_VEL
LIN {X 0,Y 350.535,Z 507.279,A -85,B 0,C 180,E1 -18613.918,E2 -18613.918} C_VEL
LIN {X 0,Y 355.954,Z 511.406,A -85,B 0,C 180,E1 -18615.477,E2 -18615.477} C_VEL
LIN {X 0,Y 361.204,Z 514.648,A -85,B 0,C 180,E1 -18617.121,E2 -18617.121} C_VEL
LIN {X 0,Y 364.576,Z 516.685,A -85,B 0,C 180,E1 -18618.33,E2 -18618.33} C_VEL
LIN {X 0,Y 368.885,Z 520.069,A -85,B 0,C 180,E1 -18620.127,E2 -18620.127} C_VEL
LIN {X 0,Y 372.366,Z 522.278,A -85,B 0,C 180,E1 -18621.851,E2 -18621.851} C_VEL
LIN {X 0,Y 375.376,Z 523.89,A -85,B 0,C 180,E1 -18623.706,E2 -18623.706} C_VEL
LIN {X 0,Y 377.255,Z 524.685,A -85,B 0,C 180,E1 -18625.198,E2 -18625.198} C_VEL
LIN {X 0,Y 379.058,Z 525.315,A -85,B 0,C 180,E1 -18627.294,E2 -18627.294} C_VEL
LIN {X 0,Y 379.744,Z 525.735,A -85,B 0,C 180,E1 -18628.939,E2 -18628.939} C_VEL
LIN {X 0,Y 379.893,Z 525.67,A -85,B 0,C 180,E1 -18630,E2 -18630} C_VEL
LIN {X 0,Y 379.625,Z 525.634,A -85,B 0,C 180,E1 -18631.43,E2 -18631.43} C_VEL
LIN {X 0,Y 378.724,Z 525.104,A -85,B 0,C 180,E1 -18633.191,E2 -18633.191} C_VEL
LIN {X 0,Y 376.927,Z 524.585,A -85,B 0,C 180,E1 -18635.077,E2 -18635.077} C_VEL
LIN {X 0,Y 374.039,Z 523.215,A -85,B 0,C 180,E1 -18637.173,E2 -18637.173} C_VEL
LIN {X 0,Y 370.602,Z 521.219,A -85,B 0,C 180,E1 -18639.06,E2 -18639.06} C_VEL
LIN {X 0,Y 366.625,Z 518.397,A -85,B 0,C 180,E1 -18640.847,E2 -18640.847} C_VEL
LIN {X 0,Y 363.236,Z 515.753,A -85,B 0,C 180,E1 -18642.174,E2 -18642.174} C_VEL
LIN {X 0,Y 358.362,Z 512.956,A -85,B 0,C 180,E1 -18643.8,E2 -18643.8} C_VEL
LIN {X 0,Y 352.644,Z 508.937,A -85,B 0,C 180,E1 -18645.49,E2 -18645.49} C_VEL
LIN {X 0,Y 347.48,Z 505.07,A -85,B 0,C 180,E1 -18646.873,E2 -18646.873} C_VEL
LIN {X 0,Y 341.291,Z 500.647,A -85,B 0,C 180,E1 -18648.373,E2 -18648.373} C_VEL
LIN {X 0,Y 334.883,Z 495.6,A -85,B 0,C 180,E1 -18649.797,E2 -18649.797} C_VEL
LIN {X 0,Y 327.595,Z 489.801,A -85,B 0,C 180,E1 -18651.269,E2 -18651.269} C_VEL
LIN {X 0,Y 318.868,Z 482.616,A -85,B 0,C 180,E1 -18652.822,E2 -18652.822} C_VEL
LIN {X 0,Y 311.048,Z 475.794,A -85,B 0,C 180,E1 -18654.036,E2 -18654.036} C_VEL
LIN {X 0,Y 301.84,Z 467.44,A -85,B 0,C 180,E1 -18655.267,E2 -18655.267} C_VEL
LIN {X 0,Y 287.708,Z 453.067,A -85,B 0,C 180,E1 -18657.023,E2 -18657.023} C_VEL
LIN {X 0,Y 279.306,Z 442.82,A -85,B 0,C 180,E1 -18658.206,E2 -18658.206} C_VEL
LIN {X 0,Y 272.149,Z 432.418,A -85,B 0,C 180,E1 -18659.332,E2 -18659.332} C_VEL
LIN {X 0,Y 259.581,Z 409.138,A -85,B 0,C 180,E1 -18661.656,E2 -18661.656} C_VEL
LIN {X 0,Y 256.312,Z 403.159,A -85,B 0,C 180,E1 -18662.335,E2 -18662.335} C_VEL
LIN {X 0,Y 256.096,Z 402.196,A -85,B 0,C 180,E1 -18662.659,E2 -18662.659} C_VEL
LIN {X 0,Y 256.116,Z 402.044,A -85,B 0,C 180,E1 -18665.186,E2 -18665.186} C_VEL
LIN {X 0,Y 256.083,Z 402.066,A -85,B 0,C 180,E1 -18669.139,E2 -18669.139} C_VEL
LIN {X 0,Y 256.06,Z 402.036,A -85,B 0,C 180,E1 -18673.326,E2 -18673.326} C_VEL
LIN {X 0,Y 256.104,Z 402.074,A -85,B 0,C 180,E1 -18677.809,E2 -18677.809} C_VEL
LIN {X 0,Y 256.094,Z 402.076,A -85,B 0,C 180,E1 -18680.863,E2 -18680.863} C_VEL
LIN {X 0,Y 256.116,Z 402.059,A -85,B 0,C 180,E1 -18684.814,E2 -18684.814} C_VEL
LIN {X 0,Y 256.087,Z 402.088,A -85,B 0,C 180,E1 -18688.573,E2 -18688.573} C_VEL
LIN {X 0,Y 256.136,Z 402.05,A -85,B 0,C 180,E1 -18692.197,E2 -18692.197} C_VEL
LIN {X 0,Y 256.162,Z 402.074,A -85,B 0,C 180,E1 -18695.7,E2 -18695.7} C_VEL
LIN {X 0,Y 256.161,Z 402.053,A -85,B 0,C 180,E1 -18699.105,E2 -18699.105} C_VEL
LIN {X 0,Y 256.295,Z 402.055,A -85,B 0,C 180,E1 -18704.086,E2 -18704.086} C_VEL
LIN {X 0,Y 256.305,Z 402.021,A -85,B 0,C 180,E1 -18708.935,E2 -18708.935} C_VEL
LIN {X 0,Y 256.535,Z 402.01,A -85,B 0,C 180,E1 -18712.128,E2 -18712.128} C_VEL
LIN {X 0,Y 256.71,Z 401.969,A -85,B 0,C 180,E1 -18718.432,E2 -18718.432} C_VEL
LIN {X 0,Y 256.71,Z 401.981,A -85,B 0,C 180,E1 -18721.57,E2 -18721.57} C_VEL
LIN {X 0,Y 256.536,Z 401.995,A -85,B 0,C 180,E1 -18727.874,E2 -18727.874} C_VEL
LIN {X 0,Y 256.306,Z 402.026,A -85,B 0,C 180,E1 -18731.067,E2 -18731.067} C_VEL
LIN {X 0,Y 256.296,Z 402.044,A -85,B 0,C 180,E1 -18735.916,E2 -18735.916} C_VEL
LIN {X 0,Y 256.164,Z 402.059,A -85,B 0,C 180,E1 -18740.896,E2 -18740.896} C_VEL
LIN {X 0,Y 256.186,Z 402.052,A -85,B 0,C 180,E1 -18745.14,E2 -18745.14} C_VEL
LIN {X 0,Y 256.112,Z 402.079,A -85,B 0,C 180,E1 -18749.601,E2 -18749.601} C_VEL
LIN {X 0,Y 256.084,Z 402.063,A -85,B 0,C 180,E1 -18753.291,E2 -18753.291} C_VEL
LIN {X 0,Y 256.141,Z 402.079,A -85,B 0,C 180,E1 -18757.28,E2 -18757.28} C_VEL
LIN {X 0,Y 256.13,Z 402.073,A -85,B 0,C 180,E1 -18761.19,E2 -18761.19} C_VEL
LIN {X 0,Y 256.072,Z 402.085,A -85,B 0,C 180,E1 -18765.528,E2 -18765.528} C_VEL
LIN {X 0,Y 256.06,Z 402.086,A -85,B 0,C 180,E1 -18766.205,E2 -18766.205} C_VEL
LIN {X 0,Y 255.353,Z 402.176,A -85,B 0,C 180,E1 -18767.097,E2 -18767.097} C_VEL
LIN {X 0,Y 252.414,Z 402.513,A -85,B 0,C 180,E1 -18768.497,E2 -18768.497} C_VEL
LIN {X 0,Y 249.691,Z 403.102,A -85,B 0,C 180,E1 -18769.897,E2 -18769.897} C_VEL
LIN {X 0,Y 249.29,Z 404.151,A -85,B 0,C 180,E1 -18770.761,E2 -18770.761} C_VEL
LIN {X 0,Y 250.629,Z 409.907,A -85,B 0,C 180,E1 -18773.924,E2 -18773.924} C_VEL
LIN {X 0,Y 251.826,Z 415.875,A -85,B 0,C 180,E1 -18776.982,E2 -18776.982} C_VEL
LIN {X 0,Y 253.346,Z 419.493,A -85,B 0,C 180,E1 -18777.419,E2 -18777.419} C_VEL
LIN {X 0,Y 258.736,Z 431.574,A -85,B 0,C 180,E1 -18778.558,E2 -18778.558} C_VEL
LIN {X 0,Y 261.224,Z 438.261,A -85,B 0,C 180,E1 -18779.098,E2 -18779.098} C_VEL
LIN {X 0,Y 265.604,Z 461.576,A -85,B 0,C 180,E1 -18780.369,E2 -18780.369} C_VEL
LIN {X 0,Y 266.664,Z 468.663,A -85,B 0,C 180,E1 -18780.712,E2 -18780.712} C_VEL
LIN {X 0,Y 264.813,Z 521.823,A -85,B 0,C 180,E1 -18782.142,E2 -18782.142} C_VEL
LIN {X 0,Y 264.097,Z 532.029,A -85,B 0,C 180,E1 -18782.583,E2 -18782.583} C_VEL
LIN {X 0,Y 262.947,Z 542.17,A -85,B 0,C 180,E1 -18783.191,E2 -18783.191} C_VEL
LIN {X 0,Y 261.738,Z 551.261,A -85,B 0,C 180,E1 -18783.917,E2 -18783.917} C_VEL
LIN {X 0,Y 260.319,Z 560.404,A -85,B 0,C 180,E1 -18784.837,E2 -18784.837} C_VEL
LIN {X 0,Y 258.657,Z 569.402,A -85,B 0,C 180,E1 -18785.949,E2 -18785.949} C_VEL
LIN {X 0,Y 256.892,Z 578.126,A -85,B 0,C 180,E1 -18787.268,E2 -18787.268} C_VEL
LIN {X 0,Y 255.296,Z 585.546,A -85,B 0,C 180,E1 -18788.608,E2 -18788.608} C_VEL
LIN {X 0,Y 253.318,Z 594.341,A -85,B 0,C 180,E1 -18790.554,E2 -18790.554} C_VEL
LIN {X 0,Y 252.024,Z 600.334,A -85,B 0,C 180,E1 -18792.137,E2 -18792.137} C_VEL
LIN {X 0,Y 250.535,Z 606.645,A -85,B 0,C 180,E1 -18794.128,E2 -18794.128} C_VEL
LIN {X 0,Y 249.225,Z 611.916,A -85,B 0,C 180,E1 -18796.132,E2 -18796.132} C_VEL
LIN {X 0,Y 248.139,Z 617.012,A -85,B 0,C 180,E1 -18798.565,E2 -18798.565} C_VEL
LIN {X 0,Y 247.418,Z 620.98,A -85,B 0,C 180,E1 -18801.012,E2 -18801.012} C_VEL
LIN {X 0,Y 247.012,Z 623.918,A -85,B 0,C 180,E1 -18803.466,E2 -18803.466} C_VEL
LIN {X 0,Y 246.885,Z 625.421,A -85,B 0,C 180,E1 -18805.102,E2 -18805.102} C_VEL
LIN {X 0,Y 246.905,Z 626.951,A -85,B 0,C 180,E1 -18808.369,E2 -18808.369} C_VEL
LIN {X 0,Y 246.975,Z 627.233,A -85,B 0,C 180,E1 -18810,E2 -18810} C_VEL
LIN {X 0,Y 246.855,Z 626.352,A -85,B 0,C 180,E1 -18813.265,E2 -18813.265} C_VEL
LIN {X 0,Y 246.885,Z 625.421,A -85,B 0,C 180,E1 -18814.899,E2 -18814.899} C_VEL
LIN {X 0,Y 247.26,Z 622.069,A -85,B 0,C 180,E1 -18818.171,E2 -18818.171} C_VEL
LIN {X 0,Y 247.847,Z 618.439,A -85,B 0,C 180,E1 -18820.622,E2 -18820.622} C_VEL
LIN {X 0,Y 248.768,Z 613.704,A -85,B 0,C 180,E1 -18823.063,E2 -18823.063} C_VEL
LIN {X 0,Y 250.223,Z 607.733,A -85,B 0,C 180,E1 -18825.476,E2 -18825.476} C_VEL
LIN {X 0,Y 251.673,Z 601.642,A -85,B 0,C 180,E1 -18827.47,E2 -18827.47} C_VEL
LIN {X 0,Y 253.068,Z 595.909,A -85,B 0,C 180,E1 -18829.043,E2 -18829.043} C_VEL
LIN {X 0,Y 254.482,Z 589.242,A -85,B 0,C 180,E1 -18830.617,E2 -18830.617} C_VEL
LIN {X 0,Y 256.218,Z 581.416,A -85,B 0,C 180,E1 -18832.158,E2 -18832.158} C_VEL
LIN {X 0,Y 257.92,Z 573.335,A -85,B 0,C 180,E1 -18833.485,E2 -18833.485} C_VEL
LIN {X 0,Y 259.768,Z 563.576,A -85,B 0,C 180,E1 -18834.794,E2 -18834.794} C_VEL
LIN {X 0,Y 261.158,Z 555.187,A -85,B 0,C 180,E1 -18835.718,E2 -18835.718} C_VEL
LIN {X 0,Y 262.618,Z 544.682,A -85,B 0,C 180,E1 -18836.632,E2 -18836.632} C_VEL
LIN {X 0,Y 263.949,Z 533.686,A -85,B 0,C 180,E1 -18837.33,E2 -18837.33} C_VEL
LIN {X 0,Y 264.797,Z 523.016,A -85,B 0,C 180,E1 -18837.808,E2 -18837.808} C_VEL
LIN {X 0,Y 265.798,Z 494.36,A -85,B 0,C 180,E1 -18838.616,E2 -18838.616} C_VEL
LIN {X 0,Y 266.638,Z 468.111,A -85,B 0,C 180,E1 -18839.308,E2 -18839.308} C_VEL
LIN {X 0,Y 262.994,Z 447.16,A -85,B 0,C 180,E1 -18840.398,E2 -18840.398} C_VEL
LIN {X 0,Y 260.537,Z 435.907,A -85,B 0,C 180,E1 -18841.066,E2 -18841.066} C_VEL
LIN {X 0,Y 254.714,Z 422.548,A -85,B 0,C 180,E1 -18842.287,E2 -18842.287} C_VEL
LIN {X 0,Y 251.873,Z 416.025,A -85,B 0,C 180,E1 -18842.976,E2 -18842.976} C_VEL
LIN {X 0,Y 250.615,Z 409.904,A -85,B 0,C 180,E1 -18846.079,E2 -18846.079} C_VEL
LIN {X 0,Y 249.045,Z 403.054,A -85,B 0,C 180,E1 -18849.908,E2 -18849.908} C_VEL
LIN {X 0,Y 249.021,Z 402.952,A -85,B 0,C 180,E1 -18852.794,E2 -18852.794} C_VEL
LIN {X 0,Y 249.084,Z 402.957,A -85,B 0,C 180,E1 -18857.376,E2 -18857.376} C_VEL
LIN {X 0,Y 249.056,Z 402.954,A -85,B 0,C 180,E1 -18861.624,E2 -18861.624} C_VEL
LIN {X 0,Y 249.064,Z 402.935,A -85,B 0,C 180,E1 -18865.642,E2 -18865.642} C_VEL
LIN {X 0,Y 249.054,Z 402.962,A -85,B 0,C 180,E1 -18869.472,E2 -18869.472} C_VEL
LIN {X 0,Y 249.075,Z 402.925,A -85,B 0,C 180,E1 -18873.162,E2 -18873.162} C_VEL
LIN {X 0,Y 249.081,Z 402.955,A -85,B 0,C 180,E1 -18876.732,E2 -18876.732} C_VEL
LIN {X 0,Y 249.111,Z 402.921,A -85,B 0,C 180,E1 -18880.211,E2 -18880.211} C_VEL
LIN {X 0,Y 249.243,Z 402.917,A -85,B 0,C 180,E1 -18883.621,E2 -18883.621} C_VEL
LIN {X 0,Y 249.253,Z 402.908,A -85,B 0,C 180,E1 -18888.616,E2 -18888.616} C_VEL
LIN {X 0,Y 249.482,Z 402.868,A -85,B 0,C 180,E1 -18891.902,E2 -18891.902} C_VEL
LIN {X 0,Y 249.436,Z 402.91,A -85,B 0,C 180,E1 -18896.769,E2 -18896.769} C_VEL
LIN {X 0,Y 249.721,Z 402.833,A -85,B 0,C 180,E1 -18899.999,E2 -18899.999} C_VEL
LIN {X 0,Y 249.436,Z 402.901,A -85,B 0,C 180,E1 -18903.229,E2 -18903.229} C_VEL
LIN {X 0,Y 249.481,Z 402.883,A -85,B 0,C 180,E1 -18908.096,E2 -18908.096} C_VEL
LIN {X 0,Y 249.252,Z 402.902,A -85,B 0,C 180,E1 -18911.382,E2 -18911.382} C_VEL
LIN {X 0,Y 249.241,Z 402.931,A -85,B 0,C 180,E1 -18916.377,E2 -18916.377} C_VEL
LIN {X 0,Y 249.086,Z 402.943,A -85,B 0,C 180,E1 -18921.517,E2 -18921.517} C_VEL
LIN {X 0,Y 249.128,Z 402.938,A -85,B 0,C 180,E1 -18925.481,E2 -18925.481} C_VEL
LIN {X 0,Y 249.071,Z 402.94,A -85,B 0,C 180,E1 -18928.988,E2 -18928.988} C_VEL
LIN {X 0,Y 249.034,Z 402.959,A -85,B 0,C 180,E1 -18932.424,E2 -18932.424} C_VEL
LIN {X 0,Y 249.066,Z 402.949,A -85,B 0,C 180,E1 -18936.338,E2 -18936.338} C_VEL
LIN {X 0,Y 249.023,Z 402.946,A -85,B 0,C 180,E1 -18940.473,E2 -18940.473} C_VEL
LIN {X 0,Y 249.004,Z 402.951,A -85,B 0,C 180,E1 -18944.877,E2 -18944.877} C_VEL
LIN {X 0,Y 249.016,Z 402.906,A -85,B 0,C 180,E1 -18947.363,E2 -18947.363} C_VEL
LIN {X 0,Y 249.037,Z 402.963,A -85,B 0,C 180,E1 -18951.621,E2 -18951.621} C_VEL
LIN {X 0,Y 249.058,Z 402.922,A -85,B 0,C 180,E1 -18955.642,E2 -18955.642} C_VEL
LIN {X 0,Y 249.09,Z 403.19,A -85,B 0,C 180,E1 -18956.447,E2 -18956.447} C_VEL
LIN {X 0,Y 249.436,Z 404.5,A -85,B 0,C 180,E1 -18956.717,E2 -18956.717} C_VEL
LIN {X 0,Y 258.328,Z 420.362,A -85,B 0,C 180,E1 -18958.531,E2 -18958.531} C_VEL
LIN {X 0,Y 267.087,Z 436.784,A -85,B 0,C 180,E1 -18960.184,E2 -18960.184} C_VEL
LIN {X 0,Y 275.412,Z 448.952,A -85,B 0,C 180,E1 -18961.534,E2 -18961.534} C_VEL
LIN {X 0,Y 285.685,Z 460.961,A -85,B 0,C 180,E1 -18962.987,E2 -18962.987} C_VEL
LIN {X 0,Y 299.433,Z 474.641,A -85,B 0,C 180,E1 -18964.691,E2 -18964.691} C_VEL
LIN {X 0,Y 308.823,Z 482.93,A -85,B 0,C 180,E1 -18965.9,E2 -18965.9} C_VEL
LIN {X 0,Y 316.81,Z 489.71,A -85,B 0,C 180,E1 -18967.099,E2 -18967.099} C_VEL
LIN {X 0,Y 323.182,Z 494.787,A -85,B 0,C 180,E1 -18968.175,E2 -18968.175} C_VEL
LIN {X 0,Y 330.152,Z 500.43,A -85,B 0,C 180,E1 -18969.492,E2 -18969.492} C_VEL
LIN {X 0,Y 337.305,Z 505.853,A -85,B 0,C 180,E1 -18970.988,E2 -18970.988} C_VEL
LIN {X 0,Y 344.355,Z 510.989,A -85,B 0,C 180,E1 -18972.615,E2 -18972.615} C_VEL
LIN {X 0,Y 351.043,Z 515.876,A -85,B 0,C 180,E1 -18974.366,E2 -18974.366} C_VEL
LIN {X 0,Y 355.844,Z 519.226,A -85,B 0,C 180,E1 -18975.756,E2 -18975.756} C_VEL
LIN {X 0,Y 360.9,Z 522.195,A -85,B 0,C 180,E1 -18977.357,E2 -18977.357} C_VEL
LIN {X 0,Y 363.091,Z 523.549,A -85,B 0,C 180,E1 -18978.138,E2 -18978.138} C_VEL
LIN {X 0,Y 367.412,Z 526.871,A -85,B 0,C 180,E1 -18979.909,E2 -18979.909} C_VEL
LIN {X 0,Y 371.055,Z 529.174,A -85,B 0,C 180,E1 -18981.675,E2 -18981.675} C_VEL
LIN {X 0,Y 374.162,Z 530.807,A -85,B 0,C 180,E1 -18983.529,E2 -18983.529} C_VEL
LIN {X 0,Y 376.275,Z 531.716,A -85,B 0,C 180,E1 -18985.185,E2 -18985.185} C_VEL
LIN {X 0,Y 377.958,Z 532.267,A -85,B 0,C 180,E1 -18987.069,E2 -18987.069} C_VEL
LIN {X 0,Y 378.779,Z 532.768,A -85,B 0,C 180,E1 -18988.937,E2 -18988.937} C_VEL
LIN {X 0,Y 378.931,Z 532.701,A -85,B 0,C 180,E1 -18990,E2 -18990} C_VEL
LIN {X 0,Y 378.672,Z 532.669,A -85,B 0,C 180,E1 -18991.433,E2 -18991.433} C_VEL
LIN {X 0,Y 377.772,Z 532.13,A -85,B 0,C 180,E1 -18993.199,E2 -18993.199} C_VEL
LIN {X 0,Y 375.952,Z 531.621,A -85,B 0,C 180,E1 -18995.09,E2 -18995.09} C_VEL
LIN {X 0,Y 373.246,Z 530.358,A -85,B 0,C 180,E1 -18997.06,E2 -18997.06} C_VEL
LIN {X 0,Y 369.756,Z 528.405,A -85,B 0,C 180,E1 -18999,E2 -18999} C_VEL
LIN {X 0,Y 365.829,Z 525.703,A -85,B 0,C 180,E1 -19000.779,E2 -19000.779} C_VEL
LIN {X 0,Y 361.437,Z 522.456,A -85,B 0,C 180,E1 -19002.458,E2 -19002.458} C_VEL
LIN {X 0,Y 356.278,Z 519.523,A -85,B 0,C 180,E1 -19004.112,E2 -19004.112} C_VEL
LIN {X 0,Y 351.016,Z 515.873,A -85,B 0,C 180,E1 -19005.641,E2 -19005.641} C_VEL
LIN {X 0,Y 345.105,Z 511.491,A -85,B 0,C 180,E1 -19007.195,E2 -19007.195} C_VEL
LIN {X 0,Y 337.824,Z 506.298,A -85,B 0,C 180,E1 -19008.894,E2 -19008.894} C_VEL
LIN {X 0,Y 331.66,Z 501.547,A -85,B 0,C 180,E1 -19010.205,E2 -19010.205} C_VEL
LIN {X 0,Y 324.834,Z 496.219,A -85,B 0,C 180,E1 -19011.516,E2 -19011.516} C_VEL
LIN {X 0,Y 317.726,Z 490.491,A -85,B 0,C 180,E1 -19012.753,E2 -19012.753} C_VEL
LIN {X 0,Y 309.952,Z 483.893,A -85,B 0,C 180,E1 -19013.94,E2 -19013.94} C_VEL
LIN {X 0,Y 301.967,Z 476.784,A -85,B 0,C 180,E1 -19015.004,E2 -19015.004} C_VEL
LIN {X 0,Y 294.341,Z 469.737,A -85,B 0,C 180,E1 -19015.916,E2 -19015.916} C_VEL
LIN {X 0,Y 282.463,Z 457.445,A -85,B 0,C 180,E1 -19017.448,E2 -19017.448} C_VEL
LIN {X 0,Y 274.561,Z 447.768,A -85,B 0,C 180,E1 -19018.598,E2 -19018.598} C_VEL
LIN {X 0,Y 266.935,Z 436.599,A -85,B 0,C 180,E1 -19019.841,E2 -19019.841} C_VEL
LIN {X 0,Y 254.292,Z 412.998,A -85,B 0,C 180,E1 -19022.273,E2 -19022.273} C_VEL
LIN {X 0,Y 250.109,Z 405.877,A -85,B 0,C 180,E1 -19023.124,E2 -19023.124} C_VEL
LIN {X 0,Y 249.201,Z 403.72,A -85,B 0,C 180,E1 -19023.398,E2 -19023.398} C_VEL
LIN {X 0,Y 249.042,Z 402.989,A -85,B 0,C 180,E1 -19023.777,E2 -19023.777} C_VEL
LIN {X 0,Y 249.053,Z 402.964,A -85,B 0,C 180,E1 -19027.804,E2 -19027.804} C_VEL
LIN {X 0,Y 249.021,Z 402.915,A -85,B 0,C 180,E1 -19030.474,E2 -19030.474} C_VEL
LIN {X 0,Y 249.004,Z 402.944,A -85,B 0,C 180,E1 -19034.878,E2 -19034.878} C_VEL
LIN {X 0,Y 249.043,Z 402.96,A -85,B 0,C 180,E1 -19037.37,E2 -19037.37} C_VEL
LIN {X 0,Y 249.043,Z 402.964,A -85,B 0,C 180,E1 -19041.624,E2 -19041.624} C_VEL
LIN {X 0,Y 249.056,Z 402.936,A -85,B 0,C 180,E1 -19045.643,E2 -19045.643} C_VEL
LIN {X 0,Y 249.046,Z 402.962,A -85,B 0,C 180,E1 -19049.474,E2 -19049.474} C_VEL
LIN {X 0,Y 249.068,Z 402.93,A -85,B 0,C 180,E1 -19053.163,E2 -19053.163} C_VEL
LIN {X 0,Y 249.074,Z 402.96,A -85,B 0,C 180,E1 -19056.733,E2 -19056.733} C_VEL
LIN {X 0,Y 249.104,Z 402.919,A -85,B 0,C 180,E1 -19060.212,E2 -19060.212} C_VEL
LIN {X 0,Y 249.237,Z 402.931,A -85,B 0,C 180,E1 -19063.623,E2 -19063.623} C_VEL
LIN {X 0,Y 249.248,Z 402.902,A -85,B 0,C 180,E1 -19068.617,E2 -19068.617} C_VEL
LIN {X 0,Y 249.477,Z 402.884,A -85,B 0,C 180,E1 -19071.904,E2 -19071.904} C_VEL
LIN {X 0,Y 249.433,Z 402.902,A -85,B 0,C 180,E1 -19076.77,E2 -19076.77} C_VEL
LIN {X 0,Y 249.717,Z 402.833,A -85,B 0,C 180,E1 -19080.001,E2 -19080.001} C_VEL
LIN {X 0,Y 249.433,Z 402.911,A -85,B 0,C 180,E1 -19083.231,E2 -19083.231} C_VEL
LIN {X 0,Y 249.478,Z 402.87,A -85,B 0,C 180,E1 -19088.098,E2 -19088.098} C_VEL
LIN {X 0,Y 249.249,Z 402.909,A -85,B 0,C 180,E1 -19091.384,E2 -19091.384} C_VEL
LIN {X 0,Y 249.239,Z 402.918,A -85,B 0,C 180,E1 -19096.379,E2 -19096.379} C_VEL
LIN {X 0,Y 249.085,Z 402.95,A -85,B 0,C 180,E1 -19101.519,E2 -19101.519} C_VEL
LIN {X 0,Y 249.129,Z 402.925,A -85,B 0,C 180,E1 -19105.483,E2 -19105.483} C_VEL
LIN {X 0,Y 249.082,Z 402.947,A -85,B 0,C 180,E1 -19108.995,E2 -19108.995} C_VEL
LIN {X 0,Y 249.035,Z 402.949,A -85,B 0,C 180,E1 -19112.426,E2 -19112.426} C_VEL
LIN {X 0,Y 249.075,Z 402.955,A -85,B 0,C 180,E1 -19116.339,E2 -19116.339} C_VEL
LIN {X 0,Y 249.083,Z 402.944,A -85,B 0,C 180,E1 -19120.464,E2 -19120.464} C_VEL
LIN {X 0,Y 249.074,Z 402.958,A -85,B 0,C 180,E1 -19122.81,E2 -19122.81} C_VEL
LIN {X 0,Y 249.025,Z 402.949,A -85,B 0,C 180,E1 -19127.366,E2 -19127.366} C_VEL
LIN {X 0,Y 249.076,Z 403.172,A -85,B 0,C 180,E1 -19130.198,E2 -19130.198} C_VEL
LIN {X 0,Y 249.29,Z 404.151,A -85,B 0,C 180,E1 -19130.761,E2 -19130.761} C_VEL
LIN {X 0,Y 249.022,Z 405.825,A -85,B 0,C 180,E1 -19131.584,E2 -19131.584} C_VEL
LIN {X 0,Y 246.823,Z 408.98,A -85,B 0,C 180,E1 -19132.859,E2 -19132.859} C_VEL
LIN {X 0,Y 244.544,Z 412.144,A -85,B 0,C 180,E1 -19134.156,E2 -19134.156} C_VEL
LIN {X 0,Y 244.188,Z 413.858,A -85,B 0,C 180,E1 -19135.002,E2 -19135.002} C_VEL
LIN {X 0,Y 244.603,Z 415.846,A -85,B 0,C 180,E1 -19135.92,E2 -19135.92} C_VEL
LIN {X 0,Y 247.882,Z 422.965,A -85,B 0,C 180,E1 -19136.731,E2 -19136.731} C_VEL
LIN {X 0,Y 253.904,Z 436.644,A -85,B 0,C 180,E1 -19138.059,E2 -19138.059} C_VEL
LIN {X 0,Y 255.374,Z 440.819,A -85,B 0,C 180,E1 -19138.398,E2 -19138.398} C_VEL
LIN {X 0,Y 259.749,Z 464.476,A -85,B 0,C 180,E1 -19139.728,E2 -19139.728} C_VEL
LIN {X 0,Y 260.438,Z 470.208,A -85,B 0,C 180,E1 -19139.995,E2 -19139.995} C_VEL
LIN {X 0,Y 258.536,Z 522.23,A -85,B 0,C 180,E1 -19141.431,E2 -19141.431} C_VEL
LIN {X 0,Y 257.794,Z 532.039,A -85,B 0,C 180,E1 -19141.867,E2 -19141.867} C_VEL
LIN {X 0,Y 256.628,Z 541.975,A -85,B 0,C 180,E1 -19142.476,E2 -19142.476} C_VEL
LIN {X 0,Y 255.385,Z 551.066,A -85,B 0,C 180,E1 -19143.217,E2 -19143.217} C_VEL
LIN {X 0,Y 253.91,Z 560.209,A -85,B 0,C 180,E1 -19144.155,E2 -19144.155} C_VEL
LIN {X 0,Y 252.186,Z 569.207,A -85,B 0,C 180,E1 -19145.291,E2 -19145.291} C_VEL
LIN {X 0,Y 250.353,Z 577.931,A -85,B 0,C 180,E1 -19146.64,E2 -19146.64} C_VEL
LIN {X 0,Y 248.665,Z 585.35,A -85,B 0,C 180,E1 -19148.008,E2 -19148.008} C_VEL
LIN {X 0,Y 246.593,Z 594.145,A -85,B 0,C 180,E1 -19150.002,E2 -19150.002} C_VEL
LIN {X 0,Y 245.252,Z 600.138,A -85,B 0,C 180,E1 -19151.627,E2 -19151.627} C_VEL
LIN {X 0,Y 243.694,Z 606.449,A -85,B 0,C 180,E1 -19153.67,E2 -19153.67} C_VEL
LIN {X 0,Y 242.305,Z 611.72,A -85,B 0,C 180,E1 -19155.728,E2 -19155.728} C_VEL
LIN {X 0,Y 241.159,Z 616.817,A -85,B 0,C 180,E1 -19158.23,E2 -19158.23} C_VEL
LIN {X 0,Y 240.384,Z 620.784,A -85,B 0,C 180,E1 -19160.747,E2 -19160.747} C_VEL
LIN {X 0,Y 239.955,Z 623.723,A -85,B 0,C 180,E1 -19163.273,E2 -19163.273} C_VEL
LIN {X 0,Y 239.794,Z 625.378,A -85,B 0,C 180,E1 -19165.207,E2 -19165.207} C_VEL
LIN {X 0,Y 239.816,Z 626.756,A -85,B 0,C 180,E1 -19168.321,E2 -19168.321} C_VEL
LIN {X 0,Y 239.884,Z 627.038,A -85,B 0,C 180,E1 -19170,E2 -19170} C_VEL
LIN {X 0,Y 239.762,Z 626.157,A -85,B 0,C 180,E1 -19173.361,E2 -19173.361} C_VEL
LIN {X 0,Y 239.803,Z 625.225,A -85,B 0,C 180,E1 -19175.045,E2 -19175.045} C_VEL
LIN {X 0,Y 240.209,Z 621.873,A -85,B 0,C 180,E1 -19178.412,E2 -19178.412} C_VEL
LIN {X 0,Y 240.85,Z 618.243,A -85,B 0,C 180,E1 -19180.934,E2 -19180.934} C_VEL
LIN {X 0,Y 241.817,Z 613.507,A -85,B 0,C 180,E1 -19183.445,E2 -19183.445} C_VEL
LIN {X 0,Y 243.378,Z 607.538,A -85,B 0,C 180,E1 -19185.922,E2 -19185.922} C_VEL
LIN {X 0,Y 244.902,Z 601.446,A -85,B 0,C 180,E1 -19187.969,E2 -19187.969} C_VEL
LIN {X 0,Y 246.446,Z 595.031,A -85,B 0,C 180,E1 -19189.765,E2 -19189.765} C_VEL
LIN {X 0,Y 248.242,Z 587.196,A -85,B 0,C 180,E1 -19191.595,E2 -19191.595} C_VEL
LIN {X 0,Y 250.138,Z 579.025,A -85,B 0,C 180,E1 -19193.163,E2 -19193.163} C_VEL
LIN {X 0,Y 251.939,Z 570.514,A -85,B 0,C 180,E1 -19194.516,E2 -19194.516} C_VEL
LIN {X 0,Y 253.637,Z 561.792,A -85,B 0,C 180,E1 -19195.655,E2 -19195.655} C_VEL
LIN {X 0,Y 255.056,Z 553.024,A -85,B 0,C 180,E1 -19196.6,E2 -19196.6} C_VEL
LIN {X 0,Y 256.449,Z 543.224,A -85,B 0,C 180,E1 -19197.436,E2 -19197.436} C_VEL
LIN {X 0,Y 257.75,Z 532.857,A -85,B 0,C 180,E1 -19198.086,E2 -19198.086} C_VEL
LIN {X 0,Y 258.518,Z 523.475,A -85,B 0,C 180,E1 -19198.518,E2 -19198.518} C_VEL
LIN {X 0,Y 259.336,Z 500.654,A -85,B 0,C 180,E1 -19199.196,E2 -19199.196} C_VEL
LIN {X 0,Y 260.373,Z 468.489,A -85,B 0,C 180,E1 -19200.067,E2 -19200.067} C_VEL
LIN {X 0,Y 256.634,Z 447.15,A -85,B 0,C 180,E1 -19201.228,E2 -19201.228} C_VEL
LIN {X 0,Y 254.726,Z 438.596,A -85,B 0,C 180,E1 -19201.763,E2 -19201.763} C_VEL
LIN {X 0,Y 247.811,Z 422.813,A -85,B 0,C 180,E1 -19203.284,E2 -19203.284} C_VEL
LIN {X 0,Y 244.684,Z 415.985,A -85,B 0,C 180,E1 -19204.045,E2 -19204.045} C_VEL
LIN {X 0,Y 244.382,Z 414.746,A -85,B 0,C 180,E1 -19204.514,E2 -19204.514} C_VEL
LIN {X 0,Y 243.101,Z 408.558,A -85,B 0,C 180,E1 -19207.968,E2 -19207.968} C_VEL
LIN {X 0,Y 241.97,Z 403.9,A -85,B 0,C 180,E1 -19210.776,E2 -19210.776} C_VEL
LIN {X 0,Y 241.97,Z 403.843,A -85,B 0,C 180,E1 -19214.193,E2 -19214.193} C_VEL
LIN {X 0,Y 242.001,Z 403.84,A -85,B 0,C 180,E1 -19218.09,E2 -19218.09} C_VEL
LIN {X 0,Y 242.016,Z 403.839,A -85,B 0,C 180,E1 -19222.422,E2 -19222.422} C_VEL
LIN {X 0,Y 241.994,Z 403.816,A -85,B 0,C 180,E1 -19226.508,E2 -19226.508} C_VEL
LIN {X 0,Y 242.039,Z 403.831,A -85,B 0,C 180,E1 -19230.586,E2 -19230.586} C_VEL
LIN {X 0,Y 242.07,Z 403.801,A -85,B 0,C 180,E1 -19234.182,E2 -19234.182} C_VEL
LIN {X 0,Y 242.055,Z 403.826,A -85,B 0,C 180,E1 -19238.296,E2 -19238.296} C_VEL
LIN {X 0,Y 242.164,Z 403.792,A -85,B 0,C 180,E1 -19243.277,E2 -19243.277} C_VEL
LIN {X 0,Y 242.187,Z 403.794,A -85,B 0,C 180,E1 -19248.279,E2 -19248.279} C_VEL
LIN {X 0,Y 242.429,Z 403.743,A -85,B 0,C 180,E1 -19251.665,E2 -19251.665} C_VEL
LIN {X 0,Y 242.261,Z 403.807,A -85,B 0,C 180,E1 -19255.006,E2 -19255.006} C_VEL
LIN {X 0,Y 242.636,Z 403.733,A -85,B 0,C 180,E1 -19258.339,E2 -19258.339} C_VEL
LIN {X 0,Y 242.636,Z 403.721,A -85,B 0,C 180,E1 -19261.659,E2 -19261.659} C_VEL
LIN {X 0,Y 242.427,Z 403.78,A -85,B 0,C 180,E1 -19266.743,E2 -19266.743} C_VEL
LIN {X 0,Y 242.313,Z 403.757,A -85,B 0,C 180,E1 -19270.021,E2 -19270.021} C_VEL
LIN {X 0,Y 242.166,Z 403.821,A -85,B 0,C 180,E1 -19275.14,E2 -19275.14} C_VEL
LIN {X 0,Y 242.071,Z 403.794,A -85,B 0,C 180,E1 -19278.623,E2 -19278.623} C_VEL
LIN {X 0,Y 242.011,Z 403.832,A -85,B 0,C 180,E1 -19282.179,E2 -19282.179} C_VEL
LIN {X 0,Y 242.065,Z 403.812,A -85,B 0,C 180,E1 -19285.837,E2 -19285.837} C_VEL
LIN {X 0,Y 242.005,Z 403.828,A -85,B 0,C 180,E1 -19289.582,E2 -19289.582} C_VEL
LIN {X 0,Y 241.989,Z 403.821,A -85,B 0,C 180,E1 -19293.49,E2 -19293.49} C_VEL
LIN {X 0,Y 242,Z 403.843,A -85,B 0,C 180,E1 -19297.579,E2 -19297.579} C_VEL
LIN {X 0,Y 241.941,Z 403.834,A -85,B 0,C 180,E1 -19301.92,E2 -19301.92} C_VEL
LIN {X 0,Y 241.934,Z 403.794,A -85,B 0,C 180,E1 -19306.57,E2 -19306.57} C_VEL
LIN {X 0,Y 241.97,Z 403.805,A -85,B 0,C 180,E1 -19310.284,E2 -19310.284} C_VEL
LIN {X 0,Y 242.034,Z 403.799,A -85,B 0,C 180,E1 -19314.497,E2 -19314.497} C_VEL
LIN {X 0,Y 242.077,Z 404.079,A -85,B 0,C 180,E1 -19315.364,E2 -19315.364} C_VEL
LIN {X 0,Y 242.434,Z 405.42,A -85,B 0,C 180,E1 -19315.648,E2 -19315.648} C_VEL
LIN {X 0,Y 251.689,Z 421.611,A -85,B 0,C 180,E1 -19317.636,E2 -19317.636} C_VEL
LIN {X 0,Y 261.651,Z 440.568,A -85,B 0,C 180,E1 -19319.612,E2 -19319.612} C_VEL
LIN {X 0,Y 269.5,Z 452.257,A -85,B 0,C 180,E1 -19320.944,E2 -19320.944} C_VEL
LIN {X 0,Y 278.15,Z 462.888,A -85,B 0,C 180,E1 -19322.241,E2 -19322.241} C_VEL
LIN {X 0,Y 289.648,Z 474.798,A -85,B 0,C 180,E1 -19323.765,E2 -19323.765} C_VEL
LIN {X 0,Y 298.308,Z 482.843,A -85,B 0,C 180,E1 -19324.8,E2 -19324.8} C_VEL
LIN {X 0,Y 307.139,Z 490.452,A -85,B 0,C 180,E1 -19325.909,E2 -19325.909} C_VEL
LIN {X 0,Y 315.275,Z 497.29,A -85,B 0,C 180,E1 -19327.105,E2 -19327.105} C_VEL
LIN {X 0,Y 322.785,Z 503.173,A -85,B 0,C 180,E1 -19328.352,E2 -19328.352} C_VEL
LIN {X 0,Y 330.125,Z 508.722,A -85,B 0,C 180,E1 -19329.739,E2 -19329.739} C_VEL
LIN {X 0,Y 338.66,Z 515.199,A -85,B 0,C 180,E1 -19331.561,E2 -19331.561} C_VEL
LIN {X 0,Y 346.187,Z 520.374,A -85,B 0,C 180,E1 -19333.372,E2 -19333.372} C_VEL
LIN {X 0,Y 352.383,Z 524.905,A -85,B 0,C 180,E1 -19335.061,E2 -19335.061} C_VEL
LIN {X 0,Y 358.276,Z 528.48,A -85,B 0,C 180,E1 -19336.87,E2 -19336.87} C_VEL
LIN {X 0,Y 361.301,Z 530.298,A -85,B 0,C 180,E1 -19337.927,E2 -19337.927} C_VEL
LIN {X 0,Y 365.802,Z 533.735,A -85,B 0,C 180,E1 -19339.774,E2 -19339.774} C_VEL
LIN {X 0,Y 369.677,Z 536.139,A -85,B 0,C 180,E1 -19341.643,E2 -19341.643} C_VEL
LIN {X 0,Y 372.793,Z 537.756,A -85,B 0,C 180,E1 -19343.505,E2 -19343.505} C_VEL
LIN {X 0,Y 374.925,Z 538.684,A -85,B 0,C 180,E1 -19345.168,E2 -19345.168} C_VEL
LIN {X 0,Y 376.632,Z 539.244,A -85,B 0,C 180,E1 -19347.058,E2 -19347.058} C_VEL
LIN {X 0,Y 377.447,Z 539.741,A -85,B 0,C 180,E1 -19348.933,E2 -19348.933} C_VEL
LIN {X 0,Y 377.609,Z 539.677,A -85,B 0,C 180,E1 -19350,E2 -19350} C_VEL
LIN {X 0,Y 377.313,Z 539.61,A -85,B 0,C 180,E1 -19351.601,E2 -19351.601} C_VEL
LIN {X 0,Y 376.473,Z 539.112,A -85,B 0,C 180,E1 -19353.21,E2 -19353.21} C_VEL
LIN {X 0,Y 374.603,Z 538.589,A -85,B 0,C 180,E1 -19355.108,E2 -19355.108} C_VEL
LIN {X 0,Y 371.873,Z 537.329,A -85,B 0,C 180,E1 -19357.086,E2 -19357.086} C_VEL
LIN {X 0,Y 368.329,Z 535.352,A -85,B 0,C 180,E1 -19359.036,E2 -19359.036} C_VEL
LIN {X 0,Y 364.45,Z 532.787,A -85,B 0,C 180,E1 -19360.8,E2 -19360.8} C_VEL
LIN {X 0,Y 359.851,Z 529.297,A -85,B 0,C 180,E1 -19362.593,E2 -19362.593} C_VEL
LIN {X 0,Y 354.312,Z 526.162,A -85,B 0,C 180,E1 -19364.366,E2 -19364.366} C_VEL
LIN {X 0,Y 347.98,Z 521.706,A -85,B 0,C 180,E1 -19366.167,E2 -19366.167} C_VEL
LIN {X 0,Y 341.942,Z 517.477,A -85,B 0,C 180,E1 -19367.678,E2 -19367.678} C_VEL
LIN {X 0,Y 334.732,Z 512.247,A -85,B 0,C 180,E1 -19369.304,E2 -19369.304} C_VEL
LIN {X 0,Y 328.167,Z 507.321,A -85,B 0,C 180,E1 -19370.646,E2 -19370.646} C_VEL
LIN {X 0,Y 321.073,Z 501.767,A -85,B 0,C 180,E1 -19371.953,E2 -19371.953} C_VEL
LIN {X 0,Y 311.864,Z 494.513,A -85,B 0,C 180,E1 -19373.422,E2 -19373.422} C_VEL
LIN {X 0,Y 302.686,Z 486.778,A -85,B 0,C 180,E1 -19374.662,E2 -19374.662} C_VEL
LIN {X 0,Y 290.51,Z 475.71,A -85,B 0,C 180,E1 -19376.126,E2 -19376.126} C_VEL
LIN {X 0,Y 277.729,Z 462.437,A -85,B 0,C 180,E1 -19377.818,E2 -19377.818} C_VEL
LIN {X 0,Y 269.742,Z 452.589,A -85,B 0,C 180,E1 -19379.018,E2 -19379.018} C_VEL
LIN {X 0,Y 261.785,Z 440.854,A -85,B 0,C 180,E1 -19380.362,E2 -19380.362} C_VEL
LIN {X 0,Y 249.284,Z 417.336,A -85,B 0,C 180,E1 -19382.862,E2 -19382.862} C_VEL
LIN {X 0,Y 243.421,Z 407.281,A -85,B 0,C 180,E1 -19384.116,E2 -19384.116} C_VEL
LIN {X 0,Y 242.175,Z 404.577,A -85,B 0,C 180,E1 -19384.481,E2 -19384.481} C_VEL
LIN {X 0,Y 242.025,Z 403.848,A -85,B 0,C 180,E1 -19384.935,E2 -19384.935} C_VEL
LIN {X 0,Y 242.003,Z 403.838,A -85,B 0,C 180,E1 -19388.364,E2 -19388.364} C_VEL
LIN {X 0,Y 241.939,Z 403.784,A -85,B 0,C 180,E1 -19391.921,E2 -19391.921} C_VEL
LIN {X 0,Y 241.975,Z 403.845,A -85,B 0,C 180,E1 -19396.56,E2 -19396.56} C_VEL
LIN {X 0,Y 241.976,Z 403.828,A -85,B 0,C 180,E1 -19400.286,E2 -19400.286} C_VEL
LIN {X 0,Y 242.031,Z 403.814,A -85,B 0,C 180,E1 -19404.498,E2 -19404.498} C_VEL
LIN {X 0,Y 241.971,Z 403.845,A -85,B 0,C 180,E1 -19408.481,E2 -19408.481} C_VEL
LIN {X 0,Y 242.003,Z 403.808,A -85,B 0,C 180,E1 -19412.313,E2 -19412.313} C_VEL
LIN {X 0,Y 242.052,Z 403.833,A -85,B 0,C 180,E1 -19416.016,E2 -19416.016} C_VEL
LIN {X 0,Y 242.031,Z 403.804,A -85,B 0,C 180,E1 -19419.608,E2 -19419.608} C_VEL
LIN {X 0,Y 242.158,Z 403.806,A -85,B 0,C 180,E1 -19423.279,E2 -19423.279} C_VEL
LIN {X 0,Y 242.182,Z 403.786,A -85,B 0,C 180,E1 -19428.281,E2 -19428.281} C_VEL
LIN {X 0,Y 242.423,Z 403.757,A -85,B 0,C 180,E1 -19431.666,E2 -19431.666} C_VEL
LIN {X 0,Y 242.258,Z 403.807,A -85,B 0,C 180,E1 -19435.008,E2 -19435.008} C_VEL
LIN {X 0,Y 242.632,Z 403.722,A -85,B 0,C 180,E1 -19438.341,E2 -19438.341} C_VEL
LIN {X 0,Y 242.633,Z 403.733,A -85,B 0,C 180,E1 -19441.661,E2 -19441.661} C_VEL
LIN {X 0,Y 242.43,Z 403.773,A -85,B 0,C 180,E1 -19446.66,E2 -19446.66} C_VEL
LIN {X 0,Y 242.311,Z 403.756,A -85,B 0,C 180,E1 -19450.023,E2 -19450.023} C_VEL
LIN {X 0,Y 242.164,Z 403.813,A -85,B 0,C 180,E1 -19455.142,E2 -19455.142} C_VEL
LIN {X 0,Y 242.07,Z 403.79,A -85,B 0,C 180,E1 -19458.625,E2 -19458.625} C_VEL
LIN {X 0,Y 242.011,Z 403.835,A -85,B 0,C 180,E1 -19462.181,E2 -19462.181} C_VEL
LIN {X 0,Y 242.065,Z 403.801,A -85,B 0,C 180,E1 -19465.839,E2 -19465.839} C_VEL
LIN {X 0,Y 242.029,Z 403.833,A -85,B 0,C 180,E1 -19469.581,E2 -19469.581} C_VEL
LIN {X 0,Y 241.99,Z 403.816,A -85,B 0,C 180,E1 -19473.492,E2 -19473.492} C_VEL
LIN {X 0,Y 242.013,Z 403.84,A -85,B 0,C 180,E1 -19477.579,E2 -19477.579} C_VEL
LIN {X 0,Y 241.998,Z 403.84,A -85,B 0,C 180,E1 -19481.911,E2 -19481.911} C_VEL
LIN {X 0,Y 241.968,Z 403.844,A -85,B 0,C 180,E1 -19486.564,E2 -19486.564} C_VEL
LIN {X 0,Y 241.996,Z 403.971,A -85,B 0,C 180,E1 -19489.343,E2 -19489.343} C_VEL
LIN {X 0,Y 243.643,Z 410.935,A -85,B 0,C 180,E1 -19493.383,E2 -19493.383} C_VEL
LIN {X 0,Y 244.188,Z 413.858,A -85,B 0,C 180,E1 -19495.002,E2 -19495.002} C_VEL
LIN {X 0,Y 244.791,Z 415.99,A -85,B 0,C 180,E1 -19495.707,E2 -19495.707} C_VEL
LIN {X 0,Y 245.759,Z 418.962,A -85,B 0,C 180,E1 -19496.212,E2 -19496.212} C_VEL
LIN {X 0,Y 247.32,Z 424.301,A -85,B 0,C 180,E1 -19496.692,E2 -19496.692} C_VEL
LIN {X 0,Y 248.577,Z 434.575,A -85,B 0,C 180,E1 -19497.213,E2 -19497.213} C_VEL
LIN {X 0,Y 249.495,Z 442.935,A -85,B 0,C 180,E1 -19497.64,E2 -19497.64} C_VEL
LIN {X 0,Y 253.739,Z 466.445,A -85,B 0,C 180,E1 -19499.003,E2 -19499.003} C_VEL
LIN {X 0,Y 254.263,Z 471.042,A -85,B 0,C 180,E1 -19499.221,E2 -19499.221} C_VEL
LIN {X 0,Y 252.359,Z 521.503,A -85,B 0,C 180,E1 -19500.64,E2 -19500.64} C_VEL
LIN {X 0,Y 251.549,Z 532.056,A -85,B 0,C 180,E1 -19501.118,E2 -19501.118} C_VEL
LIN {X 0,Y 250.374,Z 541.781,A -85,B 0,C 180,E1 -19501.727,E2 -19501.727} C_VEL
LIN {X 0,Y 249.073,Z 550.871,A -85,B 0,C 180,E1 -19502.482,E2 -19502.482} C_VEL
LIN {X 0,Y 247.536,Z 560.014,A -85,B 0,C 180,E1 -19503.439,E2 -19503.439} C_VEL
LIN {X 0,Y 245.749,Z 569.012,A -85,B 0,C 180,E1 -19504.598,E2 -19504.598} C_VEL
LIN {X 0,Y 243.857,Z 577.736,A -85,B 0,C 180,E1 -19505.979,E2 -19505.979} C_VEL
LIN {X 0,Y 242.079,Z 585.154,A -85,B 0,C 180,E1 -19507.377,E2 -19507.377} C_VEL
LIN {X 0,Y 239.89,Z 593.949,A -85,B 0,C 180,E1 -19509.418,E2 -19509.418} C_VEL
LIN {X 0,Y 238.506,Z 599.942,A -85,B 0,C 180,E1 -19511.088,E2 -19511.088} C_VEL
LIN {X 0,Y 236.865,Z 606.253,A -85,B 0,C 180,E1 -19513.185,E2 -19513.185} C_VEL
LIN {X 0,Y 235.402,Z 611.525,A -85,B 0,C 180,E1 -19515.3,E2 -19515.3} C_VEL
LIN {X 0,Y 234.172,Z 616.62,A -85,B 0,C 180,E1 -19517.873,E2 -19517.873} C_VEL
LIN {X 0,Y 233.367,Z 620.589,A -85,B 0,C 180,E1 -19520.466,E2 -19520.466} C_VEL
LIN {X 0,Y 232.892,Z 623.528,A -85,B 0,C 180,E1 -19523.068,E2 -19523.068} C_VEL
LIN {X 0,Y 232.71,Z 625.309,A -85,B 0,C 180,E1 -19525.299,E2 -19525.299} C_VEL
LIN {X 0,Y 232.729,Z 626.562,A -85,B 0,C 180,E1 -19528.27,E2 -19528.27} C_VEL
LIN {X 0,Y 232.795,Z 626.843,A -85,B 0,C 180,E1 -19530.001,E2 -19530.001} C_VEL
LIN {X 0,Y 232.671,Z 625.962,A -85,B 0,C 180,E1 -19533.464,E2 -19533.464} C_VEL
LIN {X 0,Y 232.732,Z 625.03,A -85,B 0,C 180,E1 -19535.198,E2 -19535.198} C_VEL
LIN {X 0,Y 233.177,Z 621.678,A -85,B 0,C 180,E1 -19538.668,E2 -19538.668} C_VEL
LIN {X 0,Y 233.868,Z 618.048,A -85,B 0,C 180,E1 -19541.265,E2 -19541.265} C_VEL
LIN {X 0,Y 234.881,Z 613.311,A -85,B 0,C 180,E1 -19543.85,E2 -19543.85} C_VEL
LIN {X 0,Y 236.546,Z 607.343,A -85,B 0,C 180,E1 -19546.395,E2 -19546.395} C_VEL
LIN {X 0,Y 238.147,Z 601.251,A -85,B 0,C 180,E1 -19548.497,E2 -19548.497} C_VEL
LIN {X 0,Y 239.602,Z 595.456,A -85,B 0,C 180,E1 -19550.176,E2 -19550.176} C_VEL
LIN {X 0,Y 241.189,Z 588.85,A -85,B 0,C 180,E1 -19551.81,E2 -19551.81} C_VEL
LIN {X 0,Y 243.104,Z 581.026,A -85,B 0,C 180,E1 -19553.422,E2 -19553.422} C_VEL
LIN {X 0,Y 244.916,Z 572.943,A -85,B 0,C 180,E1 -19554.814,E2 -19554.814} C_VEL
LIN {X 0,Y 246.953,Z 563.186,A -85,B 0,C 180,E1 -19556.175,E2 -19556.175} C_VEL
LIN {X 0,Y 248.424,Z 554.797,A -85,B 0,C 180,E1 -19557.141,E2 -19557.141} C_VEL
LIN {X 0,Y 250.027,Z 544.292,A -85,B 0,C 180,E1 -19558.088,E2 -19558.088} C_VEL
LIN {X 0,Y 251.407,Z 533.645,A -85,B 0,C 180,E1 -19558.795,E2 -19558.795} C_VEL
LIN {X 0,Y 252.279,Z 523.896,A -85,B 0,C 180,E1 -19559.264,E2 -19559.264} C_VEL
LIN {X 0,Y 253.094,Z 503.4,A -85,B 0,C 180,E1 -19559.895,E2 -19559.895} C_VEL
LIN {X 0,Y 254.298,Z 469.988,A -85,B 0,C 180,E1 -19560.808,E2 -19560.808} C_VEL
LIN {X 0,Y 250.808,Z 449.618,A -85,B 0,C 180,E1 -19561.951,E2 -19561.951} C_VEL
LIN {X 0,Y 249.006,Z 441.431,A -85,B 0,C 180,E1 -19562.481,E2 -19562.481} C_VEL
LIN {X 0,Y 242.562,Z 426.614,A -85,B 0,C 180,E1 -19563.963,E2 -19563.963} C_VEL
LIN {X 0,Y 238.304,Z 417.988,A -85,B 0,C 180,E1 -19564.96,E2 -19564.96} C_VEL
LIN {X 0,Y 237.331,Z 415.468,A -85,B 0,C 180,E1 -19565.303,E2 -19565.303} C_VEL
LIN {X 0,Y 236.03,Z 409.42,A -85,B 0,C 180,E1 -19568.704,E2 -19568.704} C_VEL
LIN {X 0,Y 234.918,Z 404.789,A -85,B 0,C 180,E1 -19571.588,E2 -19571.588} C_VEL
LIN {X 0,Y 234.948,Z 404.707,A -85,B 0,C 180,E1 -19575.882,E2 -19575.882} C_VEL
LIN {X 0,Y 234.958,Z 404.708,A -85,B 0,C 180,E1 -19578.847,E2 -19578.847} C_VEL
LIN {X 0,Y 234.949,Z 404.719,A -85,B 0,C 180,E1 -19583.254,E2 -19583.254} C_VEL
LIN {X 0,Y 234.963,Z 404.698,A -85,B 0,C 180,E1 -19587.424,E2 -19587.424} C_VEL
LIN {X 0,Y 234.953,Z 404.699,A -85,B 0,C 180,E1 -19591.405,E2 -19591.405} C_VEL
LIN {X 0,Y 234.989,Z 404.695,A -85,B 0,C 180,E1 -19595.246,E2 -19595.246} C_VEL
LIN {X 0,Y 235.013,Z 404.694,A -85,B 0,C 180,E1 -19598.969,E2 -19598.969} C_VEL
LIN {X 0,Y 235.097,Z 404.668,A -85,B 0,C 180,E1 -19603.059,E2 -19603.059} C_VEL
LIN {X 0,Y 235.148,Z 404.677,A -85,B 0,C 180,E1 -19607.923,E2 -19607.923} C_VEL
LIN {X 0,Y 235.378,Z 404.619,A -85,B 0,C 180,E1 -19611.413,E2 -19611.413} C_VEL
LIN {X 0,Y 235.405,Z 404.641,A -85,B 0,C 180,E1 -19613.14,E2 -19613.14} C_VEL
LIN {X 0,Y 235.596,Z 404.609,A -85,B 0,C 180,E1 -19618.29,E2 -19618.29} C_VEL
LIN {X 0,Y 235.596,Z 404.598,A -85,B 0,C 180,E1 -19621.708,E2 -19621.708} C_VEL
LIN {X 0,Y 235.404,Z 404.652,A -85,B 0,C 180,E1 -19626.858,E2 -19626.858} C_VEL
LIN {X 0,Y 235.237,Z 404.638,A -85,B 0,C 180,E1 -19630.325,E2 -19630.325} C_VEL
LIN {X 0,Y 235.113,Z 404.695,A -85,B 0,C 180,E1 -19635.605,E2 -19635.605} C_VEL
LIN {X 0,Y 235.007,Z 404.672,A -85,B 0,C 180,E1 -19639.205,E2 -19639.205} C_VEL
LIN {X 0,Y 234.96,Z 404.716,A -85,B 0,C 180,E1 -19642.882,E2 -19642.882} C_VEL
LIN {X 0,Y 234.966,Z 404.686,A -85,B 0,C 180,E1 -19646.657,E2 -19646.657} C_VEL
LIN {X 0,Y 234.921,Z 404.722,A -85,B 0,C 180,E1 -19650.568,E2 -19650.568} C_VEL
LIN {X 0,Y 234.958,Z 404.691,A -85,B 0,C 180,E1 -19654.632,E2 -19654.632} C_VEL
LIN {X 0,Y 234.939,Z 404.713,A -85,B 0,C 180,E1 -19658.944,E2 -19658.944} C_VEL
LIN {X 0,Y 234.887,Z 404.728,A -85,B 0,C 180,E1 -19663.485,E2 -19663.485} C_VEL
LIN {X 0,Y 234.887,Z 404.671,A -85,B 0,C 180,E1 -19666.514,E2 -19666.514} C_VEL
LIN {X 0,Y 234.952,Z 404.697,A -85,B 0,C 180,E1 -19671.085,E2 -19671.085} C_VEL
LIN {X 0,Y 235.008,Z 404.93,A -85,B 0,C 180,E1 -19674.156,E2 -19674.156} C_VEL
LIN {X 0,Y 235.261,Z 405.92,A -85,B 0,C 180,E1 -19674.444,E2 -19674.444} C_VEL
LIN {X 0,Y 236.924,Z 408.766,A -85,B 0,C 180,E1 -19674.859,E2 -19674.859} C_VEL
LIN {X 0,Y 247.645,Z 427.76,A -85,B 0,C 180,E1 -19677.245,E2 -19677.245} C_VEL
LIN {X 0,Y 256.537,Z 444.844,A -85,B 0,C 180,E1 -19679.072,E2 -19679.072} C_VEL
LIN {X 0,Y 264.568,Z 456.896,A -85,B 0,C 180,E1 -19680.486,E2 -19680.486} C_VEL
LIN {X 0,Y 273.21,Z 467.643,A -85,B 0,C 180,E1 -19681.829,E2 -19681.829} C_VEL
LIN {X 0,Y 285.23,Z 480.167,A -85,B 0,C 180,E1 -19683.472,E2 -19683.472} C_VEL
LIN {X 0,Y 294.129,Z 488.455,A -85,B 0,C 180,E1 -19684.561,E2 -19684.561} C_VEL
LIN {X 0,Y 303.449,Z 496.398,A -85,B 0,C 180,E1 -19685.672,E2 -19685.672} C_VEL
LIN {X 0,Y 313.242,Z 504.378,A -85,B 0,C 180,E1 -19687.027,E2 -19687.027} C_VEL
LIN {X 0,Y 321.422,Z 510.775,A -85,B 0,C 180,E1 -19688.387,E2 -19688.387} C_VEL
LIN {X 0,Y 330.182,Z 517.201,A -85,B 0,C 180,E1 -19690.065,E2 -19690.065} C_VEL
LIN {X 0,Y 337.611,Z 522.749,A -85,B 0,C 180,E1 -19691.688,E2 -19691.688} C_VEL
LIN {X 0,Y 343.914,Z 527.055,A -85,B 0,C 180,E1 -19693.212,E2 -19693.212} C_VEL
LIN {X 0,Y 350.169,Z 531.615,A -85,B 0,C 180,E1 -19694.92,E2 -19694.92} C_VEL
LIN {X 0,Y 356.059,Z 535.134,A -85,B 0,C 180,E1 -19696.721,E2 -19696.721} C_VEL
LIN {X 0,Y 359.111,Z 536.998,A -85,B 0,C 180,E1 -19697.776,E2 -19697.776} C_VEL
LIN {X 0,Y 363.774,Z 540.518,A -85,B 0,C 180,E1 -19699.688,E2 -19699.688} C_VEL
LIN {X 0,Y 366.923,Z 542.505,A -85,B 0,C 180,E1 -19701.186,E2 -19701.186} C_VEL
LIN {X 0,Y 369.068,Z 543.671,A -85,B 0,C 180,E1 -19702.34,E2 -19702.34} C_VEL
LIN {X 0,Y 370.865,Z 544.586,A -85,B 0,C 180,E1 -19703.471,E2 -19703.471} C_VEL
LIN {X 0,Y 372.393,Z 545.221,A -85,B 0,C 180,E1 -19704.585,E2 -19704.585} C_VEL
LIN {X 0,Y 373.641,Z 545.68,A -85,B 0,C 180,E1 -19705.685,E2 -19705.685} C_VEL
LIN {X 0,Y 374.62,Z 545.952,A -85,B 0,C 180,E1 -19706.773,E2 -19706.773} C_VEL
LIN {X 0,Y 375.258,Z 546.308,A -85,B 0,C 180,E1 -19707.853,E2 -19707.853} C_VEL
LIN {X 0,Y 375.619,Z 546.584,A -85,B 0,C 180,E1 -19708.928,E2 -19708.928} C_VEL
LIN {X 0,Y 375.784,Z 546.532,A -85,B 0,C 180,E1 -19710,E2 -19710} C_VEL
LIN {X 0,Y 375.639,Z 546.528,A -85,B 0,C 180,E1 -19711.072,E2 -19711.072} C_VEL
LIN {X 0,Y 375.268,Z 546.298,A -85,B 0,C 180,E1 -19712.146,E2 -19712.146} C_VEL
LIN {X 0,Y 374.63,Z 545.955,A -85,B 0,C 180,E1 -19713.226,E2 -19713.226} C_VEL
LIN {X 0,Y 373.577,Z 545.684,A -85,B 0,C 180,E1 -19714.393,E2 -19714.393} C_VEL
LIN {X 0,Y 372.403,Z 545.268,A -85,B 0,C 180,E1 -19715.414,E2 -19715.414} C_VEL
LIN {X 0,Y 370.889,Z 544.58,A -85,B 0,C 180,E1 -19716.528,E2 -19716.528} C_VEL
LIN {X 0,Y 368.836,Z 543.578,A -85,B 0,C 180,E1 -19717.769,E2 -19717.769} C_VEL
LIN {X 0,Y 365.365,Z 541.548,A -85,B 0,C 180,E1 -19719.584,E2 -19719.584} C_VEL
LIN {X 0,Y 361.454,Z 538.838,A -85,B 0,C 180,E1 -19721.288,E2 -19721.288} C_VEL
LIN {X 0,Y 357.584,Z 535.952,A -85,B 0,C 180,E1 -19722.772,E2 -19722.772} C_VEL
LIN {X 0,Y 351.865,Z 532.688,A -85,B 0,C 180,E1 -19724.579,E2 -19724.579} C_VEL
LIN {X 0,Y 345.756,Z 528.43,A -85,B 0,C 180,E1 -19726.305,E2 -19726.305} C_VEL
LIN {X 0,Y 339.868,Z 524.235,A -85,B 0,C 180,E1 -19727.789,E2 -19727.789} C_VEL
LIN {X 0,Y 332.359,Z 518.943,A -85,B 0,C 180,E1 -19729.476,E2 -19729.476} C_VEL
LIN {X 0,Y 325.821,Z 514.008,A -85,B 0,C 180,E1 -19730.798,E2 -19730.798} C_VEL
LIN {X 0,Y 318.178,Z 508.174,A -85,B 0,C 180,E1 -19732.183,E2 -19732.183} C_VEL
LIN {X 0,Y 310.165,Z 502.01,A -85,B 0,C 180,E1 -19733.412,E2 -19733.412} C_VEL
LIN {X 0,Y 302.138,Z 495.373,A -85,B 0,C 180,E1 -19734.485,E2 -19734.485} C_VEL
LIN {X 0,Y 288.958,Z 483.91,A -85,B 0,C 180,E1 -19736.055,E2 -19736.055} C_VEL
LIN {X 0,Y 274.626,Z 469.269,A -85,B 0,C 180,E1 -19737.964,E2 -19737.964} C_VEL
LIN {X 0,Y 265.242,Z 457.85,A -85,B 0,C 180,E1 -19739.402,E2 -19739.402} C_VEL
LIN {X 0,Y 256.874,Z 445.463,A -85,B 0,C 180,E1 -19740.863,E2 -19740.863} C_VEL
LIN {X 0,Y 249.437,Z 431.295,A -85,B 0,C 180,E1 -19742.37,E2 -19742.37} C_VEL
LIN {X 0,Y 242.087,Z 417.752,A -85,B 0,C 180,E1 -19743.963,E2 -19743.963} C_VEL
LIN {X 0,Y 236.571,Z 408.369,A -85,B 0,C 180,E1 -19745.216,E2 -19745.216} C_VEL
LIN {X 0,Y 235.129,Z 405.447,A -85,B 0,C 180,E1 -19745.647,E2 -19745.647} C_VEL
LIN {X 0,Y 234.981,Z 404.783,A -85,B 0,C 180,E1 -19745.985,E2 -19745.985} C_VEL
LIN {X 0,Y 234.936,Z 404.698,A -85,B 0,C 180,E1 -19748.944,E2 -19748.944} C_VEL
LIN {X 0,Y 234.885,Z 404.671,A -85,B 0,C 180,E1 -19753.485,E2 -19753.485} C_VEL
LIN {X 0,Y 234.95,Z 404.72,A -85,B 0,C 180,E1 -19756.53,E2 -19756.53} C_VEL
LIN {X 0,Y 234.949,Z 404.712,A -85,B 0,C 180,E1 -19761.086,E2 -19761.086} C_VEL
LIN {X 0,Y 234.955,Z 404.691,A -85,B 0,C 180,E1 -19765.367,E2 -19765.367} C_VEL
LIN {X 0,Y 234.964,Z 404.708,A -85,B 0,C 180,E1 -19770.158,E2 -19770.158} C_VEL
LIN {X 0,Y 234.989,Z 404.688,A -85,B 0,C 180,E1 -19773.794,E2 -19773.794} C_VEL
LIN {X 0,Y 235.006,Z 404.686,A -85,B 0,C 180,E1 -19778.97,E2 -19778.97} C_VEL
LIN {X 0,Y 235.091,Z 404.682,A -85,B 0,C 180,E1 -19783.06,E2 -19783.06} C_VEL
LIN {X 0,Y 235.142,Z 404.667,A -85,B 0,C 180,E1 -19787.924,E2 -19787.924} C_VEL
LIN {X 0,Y 235.372,Z 404.63,A -85,B 0,C 180,E1 -19791.415,E2 -19791.415} C_VEL
LIN {X 0,Y 235.4,Z 404.653,A -85,B 0,C 180,E1 -19793.142,E2 -19793.142} C_VEL
LIN {X 0,Y 235.592,Z 404.598,A -85,B 0,C 180,E1 -19798.292,E2 -19798.292} C_VEL
LIN {X 0,Y 235.592,Z 404.61,A -85,B 0,C 180,E1 -19801.71,E2 -19801.71} C_VEL
LIN {X 0,Y 235.401,Z 404.642,A -85,B 0,C 180,E1 -19806.86,E2 -19806.86} C_VEL
LIN {X 0,Y 235.235,Z 404.638,A -85,B 0,C 180,E1 -19810.328,E2 -19810.328} C_VEL
LIN {X 0,Y 235.111,Z 404.685,A -85,B 0,C 180,E1 -19815.608,E2 -19815.608} C_VEL
LIN {X 0,Y 235.006,Z 404.671,A -85,B 0,C 180,E1 -19819.207,E2 -19819.207} C_VEL
LIN {X 0,Y 234.959,Z 404.715,A -85,B 0,C 180,E1 -19822.884,E2 -19822.884} C_VEL
LIN {X 0,Y 234.968,Z 404.681,A -85,B 0,C 180,E1 -19826.659,E2 -19826.659} C_VEL
LIN {X 0,Y 234.931,Z 404.722,A -85,B 0,C 180,E1 -19830.569,E2 -19830.569} C_VEL
LIN {X 0,Y 234.96,Z 404.692,A -85,B 0,C 180,E1 -19834.634,E2 -19834.634} C_VEL
LIN {X 0,Y 234.966,Z 404.703,A -85,B 0,C 180,E1 -19838.953,E2 -19838.953} C_VEL
LIN {X 0,Y 234.974,Z 404.707,A -85,B 0,C 180,E1 -19843.467,E2 -19843.467} C_VEL
LIN {X 0,Y 234.945,Z 404.718,A -85,B 0,C 180,E1 -19846.529,E2 -19846.529} C_VEL
LIN {X 0,Y 234.941,Z 404.941,A -85,B 0,C 180,E1 -19848.561,E2 -19848.561} C_VEL
LIN {X 0,Y 236.485,Z 411.325,A -85,B 0,C 180,E1 -19852.429,E2 -19852.429} C_VEL
LIN {X 0,Y 237.338,Z 415.489,A -85,B 0,C 180,E1 -19854.702,E2 -19854.702} C_VEL
LIN {X 0,Y 239.075,Z 419.371,A -85,B 0,C 180,E1 -19855.218,E2 -19855.218} C_VEL
LIN {X 0,Y 246.513,Z 435.338,A -85,B 0,C 180,E1 -19856.945,E2 -19856.945} C_VEL
LIN {X 0,Y 249.495,Z 442.935,A -85,B 0,C 180,E1 -19857.64,E2 -19857.64} C_VEL
LIN {X 0,Y 250.095,Z 448.69,A -85,B 0,C 180,E1 -19857.917,E2 -19857.917} C_VEL
LIN {X 0,Y 249.655,Z 458.504,A -85,B 0,C 180,E1 -19858.18,E2 -19858.18} C_VEL
LIN {X 0,Y 248.05,Z 474.394,A -85,B 0,C 180,E1 -19858.48,E2 -19858.48} C_VEL
LIN {X 0,Y 246.166,Z 521.945,A -85,B 0,C 180,E1 -19859.855,E2 -19859.855} C_VEL
LIN {X 0,Y 245.35,Z 532.068,A -85,B 0,C 180,E1 -19860.33,E2 -19860.33} C_VEL
LIN {X 0,Y 244.165,Z 541.586,A -85,B 0,C 180,E1 -19860.941,E2 -19860.941} C_VEL
LIN {X 0,Y 242.809,Z 550.677,A -85,B 0,C 180,E1 -19861.709,E2 -19861.709} C_VEL
LIN {X 0,Y 241.204,Z 559.819,A -85,B 0,C 180,E1 -19862.684,E2 -19862.684} C_VEL
LIN {X 0,Y 239.355,Z 568.817,A -85,B 0,C 180,E1 -19863.869,E2 -19863.869} C_VEL
LIN {X 0,Y 237.373,Z 577.541,A -85,B 0,C 180,E1 -19865.28,E2 -19865.28} C_VEL
LIN {X 0,Y 235.518,Z 584.958,A -85,B 0,C 180,E1 -19866.711,E2 -19866.711} C_VEL
LIN {X 0,Y 233.226,Z 593.753,A -85,B 0,C 180,E1 -19868.802,E2 -19868.802} C_VEL
LIN {X 0,Y 231.787,Z 599.747,A -85,B 0,C 180,E1 -19870.518,E2 -19870.518} C_VEL
LIN {X 0,Y 230.029,Z 606.057,A -85,B 0,C 180,E1 -19872.67,E2 -19872.67} C_VEL
LIN {X 0,Y 228.518,Z 611.329,A -85,B 0,C 180,E1 -19874.847,E2 -19874.847} C_VEL
LIN {X 0,Y 227.206,Z 616.425,A -85,B 0,C 180,E1 -19877.496,E2 -19877.496} C_VEL
LIN {X 0,Y 226.332,Z 620.393,A -85,B 0,C 180,E1 -19880.167,E2 -19880.167} C_VEL
LIN {X 0,Y 225.824,Z 623.332,A -85,B 0,C 180,E1 -19882.85,E2 -19882.85} C_VEL
LIN {X 0,Y 225.618,Z 625.253,A -85,B 0,C 180,E1 -19885.425,E2 -19885.425} C_VEL
LIN {X 0,Y 225.625,Z 626.366,A -85,B 0,C 180,E1 -19888.216,E2 -19888.216} C_VEL
LIN {X 0,Y 225.708,Z 626.648,A -85,B 0,C 180,E1 -19890.001,E2 -19890.001} C_VEL
LIN {X 0,Y 225.584,Z 625.766,A -85,B 0,C 180,E1 -19893.573,E2 -19893.573} C_VEL
LIN {X 0,Y 225.646,Z 624.835,A -85,B 0,C 180,E1 -19895.362,E2 -19895.362} C_VEL
LIN {X 0,Y 226.136,Z 621.482,A -85,B 0,C 180,E1 -19898.94,E2 -19898.94} C_VEL
LIN {X 0,Y 226.874,Z 617.852,A -85,B 0,C 180,E1 -19901.617,E2 -19901.617} C_VEL
LIN {X 0,Y 227.965,Z 613.116,A -85,B 0,C 180,E1 -19904.279,E2 -19904.279} C_VEL
LIN {X 0,Y 229.729,Z 607.147,A -85,B 0,C 180,E1 -19906.896,E2 -19906.896} C_VEL
LIN {X 0,Y 231.016,Z 602.366,A -85,B 0,C 180,E1 -19908.629,E2 -19908.629} C_VEL
LIN {X 0,Y 232.452,Z 597.375,A -85,B 0,C 180,E1 -19910.199,E2 -19910.199} C_VEL
LIN {X 0,Y 234.578,Z 588.654,A -85,B 0,C 180,E1 -19912.457,E2 -19912.457} C_VEL
LIN {X 0,Y 236.606,Z 580.831,A -85,B 0,C 180,E1 -19914.106,E2 -19914.106} C_VEL
LIN {X 0,Y 238.495,Z 572.749,A -85,B 0,C 180,E1 -19915.529,E2 -19915.529} C_VEL
LIN {X 0,Y 240.59,Z 562.991,A -85,B 0,C 180,E1 -19916.922,E2 -19916.922} C_VEL
LIN {X 0,Y 242.115,Z 554.601,A -85,B 0,C 180,E1 -19917.909,E2 -19917.909} C_VEL
LIN {X 0,Y 243.775,Z 544.097,A -85,B 0,C 180,E1 -19918.875,E2 -19918.875} C_VEL
LIN {X 0,Y 245.199,Z 533.615,A -85,B 0,C 180,E1 -19919.584,E2 -19919.584} C_VEL
LIN {X 0,Y 246.144,Z 523.117,A -85,B 0,C 180,E1 -19920.093,E2 -19920.093} C_VEL
LIN {X 0,Y 247.122,Z 498.925,A -85,B 0,C 180,E1 -19920.836,E2 -19920.836} C_VEL
LIN {X 0,Y 248.145,Z 470.651,A -85,B 0,C 180,E1 -19921.631,E2 -19921.631} C_VEL
LIN {X 0,Y 244.372,Z 448.739,A -85,B 0,C 180,E1 -19922.92,E2 -19922.92} C_VEL
LIN {X 0,Y 243.149,Z 443.78,A -85,B 0,C 180,E1 -19923.276,E2 -19923.276} C_VEL
LIN {X 0,Y 235.848,Z 427.22,A -85,B 0,C 180,E1 -19925.039,E2 -19925.039} C_VEL
LIN {X 0,Y 231.465,Z 418.531,A -85,B 0,C 180,E1 -19926.123,E2 -19926.123} C_VEL
LIN {X 0,Y 230.087,Z 415.235,A -85,B 0,C 180,E1 -19926.59,E2 -19926.59} C_VEL
LIN {X 0,Y 229.249,Z 411.428,A -85,B 0,C 180,E1 -19928.777,E2 -19928.777} C_VEL
LIN {X 0,Y 227.866,Z 405.675,A -85,B 0,C 180,E1 -19932.493,E2 -19932.493} C_VEL
LIN {X 0,Y 227.92,Z 405.593,A -85,B 0,C 180,E1 -19937.282,E2 -19937.282} C_VEL
LIN {X 0,Y 227.874,Z 405.595,A -85,B 0,C 180,E1 -19941.914,E2 -19941.914} C_VEL
LIN {X 0,Y 227.893,Z 405.57,A -85,B 0,C 180,E1 -19946.372,E2 -19946.372} C_VEL
LIN {X 0,Y 227.921,Z 405.59,A -85,B 0,C 180,E1 -19950.437,E2 -19950.437} C_VEL
LIN {X 0,Y 227.931,Z 405.562,A -85,B 0,C 180,E1 -19954.425,E2 -19954.425} C_VEL
LIN {X 0,Y 227.964,Z 405.581,A -85,B 0,C 180,E1 -19958.286,E2 -19958.286} C_VEL
LIN {X 0,Y 228.036,Z 405.543,A -85,B 0,C 180,E1 -19962.825,E2 -19962.825} C_VEL
LIN {X 0,Y 228.095,Z 405.558,A -85,B 0,C 180,E1 -19967.543,E2 -19967.543} C_VEL
LIN {X 0,Y 228.307,Z 405.497,A -85,B 0,C 180,E1 -19971.145,E2 -19971.145} C_VEL
LIN {X 0,Y 228.356,Z 405.513,A -85,B 0,C 180,E1 -19972.928,E2 -19972.928} C_VEL
LIN {X 0,Y 228.555,Z 405.486,A -85,B 0,C 180,E1 -19978.237,E2 -19978.237} C_VEL
